LIN {X 0,Y 375.925,Z 316.158,A -85,B 0,C 180,E1 -12375.269,E2 -12375.269} C_VEL
LIN {X 0,Y 375.933,Z 316.15,A -85,B 0,C 180,E1 -12378.4,E2 -12378.4} C_VEL
LIN {X 0,Y 375.971,Z 316.15,A -85,B 0,C 180,E1 -12381.73,E2 -12381.73} C_VEL
LIN {X 0,Y 375.979,Z 316.144,A -85,B 0,C 180,E1 -12385.333,E2 -12385.333} C_VEL
LIN {X 0,Y 375.957,Z 316.149,A -85,B 0,C 180,E1 -12388.438,E2 -12388.438} C_VEL
LIN {X 0,Y 375.983,Z 316.148,A -85,B 0,C 180,E1 -12392.141,E2 -12392.141} C_VEL
LIN {X 0,Y 376.006,Z 316.148,A -85,B 0,C 180,E1 -12394.539,E2 -12394.539} C_VEL
LIN {X 0,Y 375.963,Z 316.147,A -85,B 0,C 180,E1 -12398.046,E2 -12398.046} C_VEL
LIN {X 0,Y 376.024,Z 316.138,A -85,B 0,C 180,E1 -12401.474,E2 -12401.474} C_VEL
LIN {X 0,Y 376.059,Z 316.138,A -85,B 0,C 180,E1 -12404.833,E2 -12404.833} C_VEL
LIN {X 0,Y 376.052,Z 316.142,A -85,B 0,C 180,E1 -12408.137,E2 -12408.137} C_VEL
LIN {X 0,Y 376.259,Z 316.11,A -85,B 0,C 180,E1 -12411.877,E2 -12411.877} C_VEL
LIN {X 0,Y 376.173,Z 316.121,A -85,B 0,C 180,E1 -12414.64,E2 -12414.64} C_VEL
LIN {X 0,Y 376.355,Z 316.102,A -85,B 0,C 180,E1 -12417.86,E2 -12417.86} C_VEL
LIN {X 0,Y 376.491,Z 316.083,A -85,B 0,C 180,E1 -12420,E2 -12420} C_VEL
LIN {X 0,Y 376.19,Z 316.122,A -85,B 0,C 180,E1 -12423.213,E2 -12423.213} C_VEL
LIN {X 0,Y 376.238,Z 316.115,A -85,B 0,C 180,E1 -12426.605,E2 -12426.605} C_VEL
LIN {X 0,Y 376.207,Z 316.119,A -85,B 0,C 180,E1 -12428.595,E2 -12428.595} C_VEL
LIN {X 0,Y 376.052,Z 316.137,A -85,B 0,C 180,E1 -12431.864,E2 -12431.864} C_VEL
LIN {X 0,Y 376.06,Z 316.141,A -85,B 0,C 180,E1 -12435.168,E2 -12435.168} C_VEL
LIN {X 0,Y 376.01,Z 316.143,A -85,B 0,C 180,E1 -12438.527,E2 -12438.527} C_VEL
LIN {X 0,Y 375.958,Z 316.153,A -85,B 0,C 180,E1 -12441.955,E2 -12441.955} C_VEL
LIN {X 0,Y 375.978,Z 316.15,A -85,B 0,C 180,E1 -12445.463,E2 -12445.463} C_VEL
LIN {X 0,Y 375.958,Z 316.156,A -85,B 0,C 180,E1 -12449.08,E2 -12449.08} C_VEL
LIN {X 0,Y 375.95,Z 316.158,A -85,B 0,C 180,E1 -12452.829,E2 -12452.829} C_VEL
LIN {X 0,Y 375.958,Z 316.155,A -85,B 0,C 180,E1 -12455.416,E2 -12455.416} C_VEL
LIN {X 0,Y 375.975,Z 316.15,A -85,B 0,C 180,E1 -12458.271,E2 -12458.271} C_VEL
LIN {X 0,Y 376.009,Z 316.268,A -85,B 0,C 180,E1 -12459.974,E2 -12459.974} C_VEL
LIN {X 0,Y 378.221,Z 326.76,A -85,B 0,C 180,E1 -12462.706,E2 -12462.706} C_VEL
LIN {X 0,Y 378.98,Z 330.682,A -85,B 0,C 180,E1 -12463.678,E2 -12463.678} C_VEL
LIN {X 0,Y 378.967,Z 334.995,A -85,B 0,C 180,E1 -12464.597,E2 -12464.597} C_VEL
LIN {X 0,Y 383.33,Z 356.245,A -85,B 0,C 180,E1 -12465.33,E2 -12465.33} C_VEL
LIN {X 0,Y 384.181,Z 362.884,A -85,B 0,C 180,E1 -12465.516,E2 -12465.516} C_VEL
LIN {X 0,Y 382.729,Z 441.201,A -85,B 0,C 180,E1 -12467.044,E2 -12467.044} C_VEL
LIN {X 0,Y 382.323,Z 451.45,A -85,B 0,C 180,E1 -12467.361,E2 -12467.361} C_VEL
LIN {X 0,Y 381.894,Z 461.344,A -85,B 0,C 180,E1 -12467.801,E2 -12467.801} C_VEL
LIN {X 0,Y 381.198,Z 471.819,A -85,B 0,C 180,E1 -12468.416,E2 -12468.416} C_VEL
LIN {X 0,Y 380.503,Z 481.268,A -85,B 0,C 180,E1 -12469.119,E2 -12469.119} C_VEL
LIN {X 0,Y 379.709,Z 490.561,A -85,B 0,C 180,E1 -12469.97,E2 -12469.97} C_VEL
LIN {X 0,Y 378.669,Z 500.677,A -85,B 0,C 180,E1 -12471.115,E2 -12471.115} C_VEL
LIN {X 0,Y 377.901,Z 508.256,A -85,B 0,C 180,E1 -12472.141,E2 -12472.141} C_VEL
LIN {X 0,Y 377.111,Z 515.955,A -85,B 0,C 180,E1 -12473.39,E2 -12473.39} C_VEL
LIN {X 0,Y 376.23,Z 524.101,A -85,B 0,C 180,E1 -12475.019,E2 -12475.019} C_VEL
LIN {X 0,Y 375.749,Z 529.029,A -85,B 0,C 180,E1 -12476.19,E2 -12476.19} C_VEL
LIN {X 0,Y 375.202,Z 534.748,A -85,B 0,C 180,E1 -12477.882,E2 -12477.882} C_VEL
LIN {X 0,Y 374.831,Z 539.238,A -85,B 0,C 180,E1 -12479.598,E2 -12479.598} C_VEL
LIN {X 0,Y 374.655,Z 541.781,A -85,B 0,C 180,E1 -12480.809,E2 -12480.809} C_VEL
LIN {X 0,Y 374.469,Z 543.607,A -85,B 0,C 180,E1 -12482.018,E2 -12482.018} C_VEL
LIN {X 0,Y 374.226,Z 545.847,A -85,B 0,C 180,E1 -12484.349,E2 -12484.349} C_VEL
LIN {X 0,Y 374.166,Z 546.21,A -85,B 0,C 180,E1 -12485.592,E2 -12485.592} C_VEL
LIN {X 0,Y 374.215,Z 545.984,A -85,B 0,C 180,E1 -12486.963,E2 -12486.963} C_VEL
LIN {X 0,Y 374.245,Z 545.511,A -85,B 0,C 180,E1 -12487.94,E2 -12487.94} C_VEL
LIN {X 0,Y 374.428,Z 543.566,A -85,B 0,C 180,E1 -12489.801,E2 -12489.801} C_VEL
LIN {X 0,Y 374.643,Z 540.922,A -85,B 0,C 180,E1 -12491.403,E2 -12491.403} C_VEL
LIN {X 0,Y 374.892,Z 537.413,A -85,B 0,C 180,E1 -12492.957,E2 -12492.957} C_VEL
LIN {X 0,Y 375.172,Z 533.777,A -85,B 0,C 180,E1 -12494.239,E2 -12494.239} C_VEL
LIN {X 0,Y 375.665,Z 527.744,A -85,B 0,C 180,E1 -12495.924,E2 -12495.924} C_VEL
LIN {X 0,Y 376.402,Z 520.097,A -85,B 0,C 180,E1 -12497.601,E2 -12497.601} C_VEL
LIN {X 0,Y 377.122,Z 512.342,A -85,B 0,C 180,E1 -12498.988,E2 -12498.988} C_VEL
LIN {X 0,Y 377.905,Z 504.742,A -85,B 0,C 180,E1 -12500.122,E2 -12500.122} C_VEL
LIN {X 0,Y 378.638,Z 496.199,A -85,B 0,C 180,E1 -12501.192,E2 -12501.192} C_VEL
LIN {X 0,Y 379.538,Z 486.88,A -85,B 0,C 180,E1 -12502.151,E2 -12502.151} C_VEL
LIN {X 0,Y 380.257,Z 477.25,A -85,B 0,C 180,E1 -12502.967,E2 -12502.967} C_VEL
LIN {X 0,Y 380.884,Z 467.314,A -85,B 0,C 180,E1 -12503.644,E2 -12503.644} C_VEL
LIN {X 0,Y 381.489,Z 455.363,A -85,B 0,C 180,E1 -12504.254,E2 -12504.254} C_VEL
LIN {X 0,Y 381.984,Z 444.529,A -85,B 0,C 180,E1 -12504.64,E2 -12504.64} C_VEL
LIN {X 0,Y 382.331,Z 427.037,A -85,B 0,C 180,E1 -12505.025,E2 -12505.025} C_VEL
LIN {X 0,Y 383.365,Z 360.957,A -85,B 0,C 180,E1 -12506.285,E2 -12506.285} C_VEL
LIN {X 0,Y 379.739,Z 341.554,A -85,B 0,C 180,E1 -12506.864,E2 -12506.864} C_VEL
LIN {X 0,Y 378.777,Z 338.239,A -85,B 0,C 180,E1 -12507.067,E2 -12507.067} C_VEL
LIN {X 0,Y 377.196,Z 334.864,A -85,B 0,C 180,E1 -12507.503,E2 -12507.503} C_VEL
LIN {X 0,Y 374.754,Z 331.16,A -85,B 0,C 180,E1 -12508.331,E2 -12508.331} C_VEL
LIN {X 0,Y 371.314,Z 325.692,A -85,B 0,C 180,E1 -12509.995,E2 -12509.995} C_VEL
LIN {X 0,Y 370.628,Z 323.671,A -85,B 0,C 180,E1 -12510.575,E2 -12510.575} C_VEL
LIN {X 0,Y 369.258,Z 317.027,A -85,B 0,C 180,E1 -12512.523,E2 -12512.523} C_VEL
LIN {X 0,Y 369.189,Z 316.994,A -85,B 0,C 180,E1 -12516.559,E2 -12516.559} C_VEL
LIN {X 0,Y 369.065,Z 317.013,A -85,B 0,C 180,E1 -12519.868,E2 -12519.868} C_VEL
LIN {X 0,Y 369.039,Z 317.019,A -85,B 0,C 180,E1 -12523.772,E2 -12523.772} C_VEL
LIN {X 0,Y 369.003,Z 317.022,A -85,B 0,C 180,E1 -12527.768,E2 -12527.768} C_VEL
LIN {X 0,Y 368.912,Z 317.029,A -85,B 0,C 180,E1 -12531.221,E2 -12531.221} C_VEL
LIN {X 0,Y 368.957,Z 317.026,A -85,B 0,C 180,E1 -12534.776,E2 -12534.776} C_VEL
LIN {X 0,Y 368.965,Z 317.018,A -85,B 0,C 180,E1 -12537.203,E2 -12537.203} C_VEL
LIN {X 0,Y 368.931,Z 317.029,A -85,B 0,C 180,E1 -12540.954,E2 -12540.954} C_VEL
LIN {X 0,Y 368.93,Z 317.014,A -85,B 0,C 180,E1 -12545.001,E2 -12545.001} C_VEL
LIN {X 0,Y 368.91,Z 317.028,A -85,B 0,C 180,E1 -12548.64,E2 -12548.64} C_VEL
LIN {X 0,Y 368.883,Z 317.019,A -85,B 0,C 180,E1 -12552.009,E2 -12552.009} C_VEL
LIN {X 0,Y 368.885,Z 317.032,A -85,B 0,C 180,E1 -12555.176,E2 -12555.176} C_VEL
LIN {X 0,Y 368.875,Z 317.03,A -85,B 0,C 180,E1 -12558.176,E2 -12558.176} C_VEL
LIN {X 0,Y 368.883,Z 317.019,A -85,B 0,C 180,E1 -12561.365,E2 -12561.365} C_VEL
LIN {X 0,Y 368.938,Z 317.028,A -85,B 0,C 180,E1 -12565.146,E2 -12565.146} C_VEL
LIN {X 0,Y 368.931,Z 317.015,A -85,B 0,C 180,E1 -12569.046,E2 -12569.046} C_VEL
LIN {X 0,Y 368.879,Z 317.023,A -85,B 0,C 180,E1 -12572.79,E2 -12572.79} C_VEL
LIN {X 0,Y 368.935,Z 317.029,A -85,B 0,C 180,E1 -12576.117,E2 -12576.117} C_VEL
LIN {X 0,Y 368.939,Z 317.013,A -85,B 0,C 180,E1 -12579.947,E2 -12579.947} C_VEL
LIN {X 0,Y 368.971,Z 317.006,A -85,B 0,C 180,E1 -12583.398,E2 -12583.398} C_VEL
LIN {X 0,Y 369.06,Z 317.009,A -85,B 0,C 180,E1 -12586.79,E2 -12586.79} C_VEL
LIN {X 0,Y 369.064,Z 317.002,A -85,B 0,C 180,E1 -12590.131,E2 -12590.131} C_VEL
LIN {X 0,Y 369.161,Z 316.972,A -85,B 0,C 180,E1 -12593.441,E2 -12593.441} C_VEL
LIN {X 0,Y 369.304,Z 316.976,A -85,B 0,C 180,E1 -12597.818,E2 -12597.818} C_VEL
LIN {X 0,Y 369.237,Z 316.983,A -85,B 0,C 180,E1 -12601.09,E2 -12601.09} C_VEL
LIN {X 0,Y 369.303,Z 316.976,A -85,B 0,C 180,E1 -12602.181,E2 -12602.181} C_VEL
LIN {X 0,Y 369.181,Z 316.979,A -85,B 0,C 180,E1 -12606.558,E2 -12606.558} C_VEL
LIN {X 0,Y 369.064,Z 317.01,A -85,B 0,C 180,E1 -12609.868,E2 -12609.868} C_VEL
LIN {X 0,Y 369.039,Z 316.998,A -85,B 0,C 180,E1 -12613.772,E2 -12613.772} C_VEL
LIN {X 0,Y 368.954,Z 317.019,A -85,B 0,C 180,E1 -12617.744,E2 -12617.744} C_VEL
LIN {X 0,Y 368.91,Z 317.026,A -85,B 0,C 180,E1 -12621.22,E2 -12621.22} C_VEL
LIN {X 0,Y 368.923,Z 317.018,A -85,B 0,C 180,E1 -12624.777,E2 -12624.777} C_VEL
LIN {X 0,Y 368.893,Z 317.035,A -85,B 0,C 180,E1 -12628.792,E2 -12628.792} C_VEL
LIN {X 0,Y 368.897,Z 317.023,A -85,B 0,C 180,E1 -12632.238,E2 -12632.238} C_VEL
LIN {X 0,Y 368.927,Z 317.029,A -85,B 0,C 180,E1 -12635.001,E2 -12635.001} C_VEL
LIN {X 0,Y 368.875,Z 317.031,A -85,B 0,C 180,E1 -12638.633,E2 -12638.633} C_VEL
LIN {X 0,Y 368.856,Z 317.033,A -85,B 0,C 180,E1 -12642.005,E2 -12642.005} C_VEL
LIN {X 0,Y 368.871,Z 317.033,A -85,B 0,C 180,E1 -12645.174,E2 -12645.174} C_VEL
LIN {X 0,Y 368.858,Z 317.038,A -85,B 0,C 180,E1 -12648.174,E2 -12648.174} C_VEL
LIN {X 0,Y 368.875,Z 317.034,A -85,B 0,C 180,E1 -12651.366,E2 -12651.366} C_VEL
LIN {X 0,Y 368.929,Z 317.03,A -85,B 0,C 180,E1 -12655.145,E2 -12655.145} C_VEL
LIN {X 0,Y 368.911,Z 317.028,A -85,B 0,C 180,E1 -12659.045,E2 -12659.045} C_VEL
LIN {X 0,Y 368.922,Z 317.065,A -85,B 0,C 180,E1 -12661.436,E2 -12661.436} C_VEL
LIN {X 0,Y 369.725,Z 320.883,A -85,B 0,C 180,E1 -12662.551,E2 -12662.551} C_VEL
LIN {X 0,Y 372.093,Z 333.056,A -85,B 0,C 180,E1 -12665.744,E2 -12665.744} C_VEL
LIN {X 0,Y 372.19,Z 336.68,A -85,B 0,C 180,E1 -12666.638,E2 -12666.638} C_VEL
LIN {X 0,Y 371.462,Z 345.045,A -85,B 0,C 180,E1 -12668.565,E2 -12668.565} C_VEL
LIN {X 0,Y 376.368,Z 374.14,A -85,B 0,C 180,E1 -12669.45,E2 -12669.45} C_VEL
LIN {X 0,Y 375.41,Z 443.445,A -85,B 0,C 180,E1 -12670.805,E2 -12670.805} C_VEL
LIN {X 0,Y 374.992,Z 459.033,A -85,B 0,C 180,E1 -12671.208,E2 -12671.208} C_VEL
LIN {X 0,Y 374.213,Z 471.284,A -85,B 0,C 180,E1 -12671.735,E2 -12671.735} C_VEL
LIN {X 0,Y 373.661,Z 481.522,A -85,B 0,C 180,E1 -12672.345,E2 -12672.345} C_VEL
LIN {X 0,Y 372.753,Z 492.128,A -85,B 0,C 180,E1 -12673.149,E2 -12673.149} C_VEL
LIN {X 0,Y 371.932,Z 502.076,A -85,B 0,C 180,E1 -12674.098,E2 -12674.098} C_VEL
LIN {X 0,Y 371.073,Z 511.172,A -85,B 0,C 180,E1 -12675.155,E2 -12675.155} C_VEL
LIN {X 0,Y 370.312,Z 519.206,A -85,B 0,C 180,E1 -12676.277,E2 -12676.277} C_VEL
LIN {X 0,Y 369.503,Z 527.325,A -85,B 0,C 180,E1 -12677.644,E2 -12677.644} C_VEL
LIN {X 0,Y 368.779,Z 534.078,A -85,B 0,C 180,E1 -12679.014,E2 -12679.014} C_VEL
LIN {X 0,Y 368.379,Z 538.745,A -85,B 0,C 180,E1 -12680.113,E2 -12680.113} C_VEL
LIN {X 0,Y 367.913,Z 544.422,A -85,B 0,C 180,E1 -12681.763,E2 -12681.763} C_VEL
LIN {X 0,Y 367.624,Z 548.89,A -85,B 0,C 180,E1 -12683.413,E2 -12683.413} C_VEL
LIN {X 0,Y 367.488,Z 551.209,A -85,B 0,C 180,E1 -12684.513,E2 -12684.513} C_VEL
LIN {X 0,Y 367.348,Z 554.67,A -85,B 0,C 180,E1 -12686.71,E2 -12686.71} C_VEL
LIN {X 0,Y 367.345,Z 556.31,A -85,B 0,C 180,E1 -12688.904,E2 -12688.904} C_VEL
LIN {X 0,Y 367.369,Z 556.628,A -85,B 0,C 180,E1 -12690,E2 -12690} C_VEL
LIN {X 0,Y 367.312,Z 555.904,A -85,B 0,C 180,E1 -12692.193,E2 -12692.193} C_VEL
LIN {X 0,Y 367.351,Z 554.929,A -85,B 0,C 180,E1 -12693.29,E2 -12693.29} C_VEL
LIN {X 0,Y 367.514,Z 551.83,A -85,B 0,C 180,E1 -12695.487,E2 -12695.487} C_VEL
LIN {X 0,Y 367.697,Z 548.302,A -85,B 0,C 180,E1 -12697.137,E2 -12697.137} C_VEL
LIN {X 0,Y 368.077,Z 543.676,A -85,B 0,C 180,E1 -12698.786,E2 -12698.786} C_VEL
LIN {X 0,Y 368.652,Z 537.8,A -85,B 0,C 180,E1 -12700.434,E2 -12700.434} C_VEL
LIN {X 0,Y 369.38,Z 530.442,A -85,B 0,C 180,E1 -12702.081,E2 -12702.081} C_VEL
LIN {X 0,Y 370.261,Z 522.998,A -85,B 0,C 180,E1 -12703.445,E2 -12703.445} C_VEL
LIN {X 0,Y 371.091,Z 515.106,A -85,B 0,C 180,E1 -12704.655,E2 -12704.655} C_VEL
LIN {X 0,Y 371.993,Z 506.465,A -85,B 0,C 180,E1 -12705.758,E2 -12705.758} C_VEL
LIN {X 0,Y 372.838,Z 497.564,A -85,B 0,C 180,E1 -12706.706,E2 -12706.706} C_VEL
LIN {X 0,Y 373.878,Z 486.51,A -85,B 0,C 180,E1 -12707.644,E2 -12707.644} C_VEL
LIN {X 0,Y 374.673,Z 476.626,A -85,B 0,C 180,E1 -12708.312,E2 -12708.312} C_VEL
LIN {X 0,Y 375.392,Z 465.654,A -85,B 0,C 180,E1 -12708.877,E2 -12708.877} C_VEL
LIN {X 0,Y 375.96,Z 454.848,A -85,B 0,C 180,E1 -12709.272,E2 -12709.272} C_VEL
LIN {X 0,Y 376.343,Z 437.6,A -85,B 0,C 180,E1 -12709.663,E2 -12709.663} C_VEL
LIN {X 0,Y 377.26,Z 374.153,A -85,B 0,C 180,E1 -12710.916,E2 -12710.916} C_VEL
LIN {X 0,Y 372.87,Z 349.586,A -85,B 0,C 180,E1 -12711.71,E2 -12711.71} C_VEL
LIN {X 0,Y 371.857,Z 344.362,A -85,B 0,C 180,E1 -12711.94,E2 -12711.94} C_VEL
LIN {X 0,Y 372.591,Z 335.605,A -85,B 0,C 180,E1 -12713.925,E2 -12713.925} C_VEL
LIN {X 0,Y 370.858,Z 325.957,A -85,B 0,C 180,E1 -12716.403,E2 -12716.403} C_VEL
LIN {X 0,Y 368.916,Z 317.18,A -85,B 0,C 180,E1 -12718.8,E2 -12718.8} C_VEL
LIN {X 0,Y 368.896,Z 317.032,A -85,B 0,C 180,E1 -12722.238,E2 -12722.238} C_VEL
LIN {X 0,Y 368.927,Z 317.032,A -85,B 0,C 180,E1 -12725.002,E2 -12725.002} C_VEL
LIN {X 0,Y 368.904,Z 317.035,A -85,B 0,C 180,E1 -12728.64,E2 -12728.64} C_VEL
LIN {X 0,Y 368.872,Z 317.035,A -85,B 0,C 180,E1 -12732.008,E2 -12732.008} C_VEL
LIN {X 0,Y 368.878,Z 317.037,A -85,B 0,C 180,E1 -12735.176,E2 -12735.176} C_VEL
LIN {X 0,Y 368.881,Z 317.03,A -85,B 0,C 180,E1 -12738.178,E2 -12738.178} C_VEL
LIN {X 0,Y 368.906,Z 317.03,A -85,B 0,C 180,E1 -12741.36,E2 -12741.36} C_VEL
LIN {X 0,Y 368.936,Z 317.02,A -85,B 0,C 180,E1 -12745.147,E2 -12745.147} C_VEL
LIN {X 0,Y 368.928,Z 317.024,A -85,B 0,C 180,E1 -12749.047,E2 -12749.047} C_VEL
LIN {X 0,Y 368.963,Z 317.02,A -85,B 0,C 180,E1 -12752.797,E2 -12752.797} C_VEL
LIN {X 0,Y 368.945,Z 317.023,A -85,B 0,C 180,E1 -12756.113,E2 -12756.113} C_VEL
LIN {X 0,Y 368.937,Z 317.025,A -85,B 0,C 180,E1 -12759.947,E2 -12759.947} C_VEL
LIN {X 0,Y 368.977,Z 317.024,A -85,B 0,C 180,E1 -12763.399,E2 -12763.399} C_VEL
LIN {X 0,Y 369.058,Z 317.003,A -85,B 0,C 180,E1 -12766.791,E2 -12766.791} C_VEL
LIN {X 0,Y 369.069,Z 317.005,A -85,B 0,C 180,E1 -12770.132,E2 -12770.132} C_VEL
LIN {X 0,Y 369.19,Z 316.997,A -85,B 0,C 180,E1 -12772.343,E2 -12772.343} C_VEL
LIN {X 0,Y 369.146,Z 316.998,A -85,B 0,C 180,E1 -12774.538,E2 -12774.538} C_VEL
LIN {X 0,Y 369.32,Z 316.978,A -85,B 0,C 180,E1 -12777.819,E2 -12777.819} C_VEL
LIN {X 0,Y 369.46,Z 316.958,A -85,B 0,C 180,E1 -12780,E2 -12780} C_VEL
LIN {X 0,Y 369.32,Z 316.978,A -85,B 0,C 180,E1 -12782.181,E2 -12782.181} C_VEL
LIN {X 0,Y 369.208,Z 316.992,A -85,B 0,C 180,E1 -12786.592,E2 -12786.592} C_VEL
LIN {X 0,Y 369.139,Z 316.999,A -85,B 0,C 180,E1 -12788.761,E2 -12788.761} C_VEL
LIN {X 0,Y 369.007,Z 317.013,A -85,B 0,C 180,E1 -12792.093,E2 -12792.093} C_VEL
LIN {X 0,Y 368.999,Z 317.02,A -85,B 0,C 180,E1 -12795.465,E2 -12795.465} C_VEL
LIN {X 0,Y 368.96,Z 317.02,A -85,B 0,C 180,E1 -12798.894,E2 -12798.894} C_VEL
LIN {X 0,Y 368.923,Z 317.03,A -85,B 0,C 180,E1 -12802.396,E2 -12802.396} C_VEL
LIN {X 0,Y 368.962,Z 317.026,A -85,B 0,C 180,E1 -12805.983,E2 -12805.983} C_VEL
LIN {X 0,Y 368.944,Z 317.024,A -85,B 0,C 180,E1 -12808.807,E2 -12808.807} C_VEL
LIN {X 0,Y 368.899,Z 317.031,A -85,B 0,C 180,E1 -12812.238,E2 -12812.238} C_VEL
LIN {X 0,Y 368.93,Z 317.029,A -85,B 0,C 180,E1 -12815.002,E2 -12815.002} C_VEL
LIN {X 0,Y 368.912,Z 317.03,A -85,B 0,C 180,E1 -12818.641,E2 -12818.641} C_VEL
LIN {X 0,Y 368.98,Z 317.254,A -85,B 0,C 180,E1 -12819.649,E2 -12819.649} C_VEL
LIN {X 0,Y 371.215,Z 327.729,A -85,B 0,C 180,E1 -12822.408,E2 -12822.408} C_VEL
LIN {X 0,Y 372.128,Z 333.344,A -85,B 0,C 180,E1 -12823.813,E2 -12823.813} C_VEL
LIN {X 0,Y 372.155,Z 335.145,A -85,B 0,C 180,E1 -12824.158,E2 -12824.158} C_VEL
LIN {X 0,Y 376.778,Z 357.392,A -85,B 0,C 180,E1 -12824.949,E2 -12824.949} C_VEL
LIN {X 0,Y 377.575,Z 364.271,A -85,B 0,C 180,E1 -12825.142,E2 -12825.142} C_VEL
LIN {X 0,Y 376.088,Z 441.078,A -85,B 0,C 180,E1 -12826.667,E2 -12826.667} C_VEL
LIN {X 0,Y 375.682,Z 450.833,A -85,B 0,C 180,E1 -12826.964,E2 -12826.964} C_VEL
LIN {X 0,Y 375.204,Z 461.645,A -85,B 0,C 180,E1 -12827.453,E2 -12827.453} C_VEL
LIN {X 0,Y 374.499,Z 471.624,A -85,B 0,C 180,E1 -12828.045,E2 -12828.045} C_VEL
LIN {X 0,Y 373.69,Z 481.951,A -85,B 0,C 180,E1 -12828.834,E2 -12828.834} C_VEL
LIN {X 0,Y 372.786,Z 491.886,A -85,B 0,C 180,E1 -12829.782,E2 -12829.782} C_VEL
LIN {X 0,Y 371.846,Z 500.671,A -85,B 0,C 180,E1 -12830.797,E2 -12830.797} C_VEL
LIN {X 0,Y 370.924,Z 509.201,A -85,B 0,C 180,E1 -12831.991,E2 -12831.991} C_VEL
LIN {X 0,Y 370.106,Z 516.757,A -85,B 0,C 180,E1 -12833.262,E2 -12833.262} C_VEL
LIN {X 0,Y 369.286,Z 524.062,A -85,B 0,C 180,E1 -12834.753,E2 -12834.753} C_VEL
LIN {X 0,Y 368.707,Z 529.598,A -85,B 0,C 180,E1 -12836.114,E2 -12836.114} C_VEL
LIN {X 0,Y 368.192,Z 534.815,A -85,B 0,C 180,E1 -12837.693,E2 -12837.693} C_VEL
LIN {X 0,Y 367.783,Z 539.033,A -85,B 0,C 180,E1 -12839.307,E2 -12839.307} C_VEL
LIN {X 0,Y 367.566,Z 542.088,A -85,B 0,C 180,E1 -12840.819,E2 -12840.819} C_VEL
LIN {X 0,Y 367.26,Z 544.621,A -85,B 0,C 180,E1 -12842.66,E2 -12842.66} C_VEL
LIN {X 0,Y 367.132,Z 545.87,A -85,B 0,C 180,E1 -12844.122,E2 -12844.122} C_VEL
LIN {X 0,Y 367.101,Z 546.282,A -85,B 0,C 180,E1 -12846.295,E2 -12846.295} C_VEL
LIN {X 0,Y 367.144,Z 545.926,A -85,B 0,C 180,E1 -12847.49,E2 -12847.49} C_VEL
LIN {X 0,Y 367.343,Z 543.661,A -85,B 0,C 180,E1 -12849.856,E2 -12849.856} C_VEL
LIN {X 0,Y 367.586,Z 540.758,A -85,B 0,C 180,E1 -12851.611,E2 -12851.611} C_VEL
LIN {X 0,Y 367.785,Z 538.147,A -85,B 0,C 180,E1 -12852.834,E2 -12852.834} C_VEL
LIN {X 0,Y 368.143,Z 533.493,A -85,B 0,C 180,E1 -12854.498,E2 -12854.498} C_VEL
LIN {X 0,Y 368.773,Z 526.54,A -85,B 0,C 180,E1 -12856.397,E2 -12856.397} C_VEL
LIN {X 0,Y 369.334,Z 521.038,A -85,B 0,C 180,E1 -12857.639,E2 -12857.639} C_VEL
LIN {X 0,Y 370.062,Z 513.447,A -85,B 0,C 180,E1 -12859.052,E2 -12859.052} C_VEL
LIN {X 0,Y 370.962,Z 504.768,A -85,B 0,C 180,E1 -12860.378,E2 -12860.378} C_VEL
LIN {X 0,Y 371.742,Z 496.455,A -85,B 0,C 180,E1 -12861.438,E2 -12861.438} C_VEL
LIN {X 0,Y 372.661,Z 487.172,A -85,B 0,C 180,E1 -12862.414,E2 -12862.414} C_VEL
LIN {X 0,Y 373.416,Z 477.576,A -85,B 0,C 180,E1 -12863.245,E2 -12863.245} C_VEL
LIN {X 0,Y 374.195,Z 466.065,A -85,B 0,C 180,E1 -12864.023,E2 -12864.023} C_VEL
LIN {X 0,Y 374.726,Z 455.366,A -85,B 0,C 180,E1 -12864.573,E2 -12864.573} C_VEL
LIN {X 0,Y 375.214,Z 444.628,A -85,B 0,C 180,E1 -12864.963,E2 -12864.963} C_VEL
LIN {X 0,Y 375.575,Z 427.978,A -85,B 0,C 180,E1 -12865.338,E2 -12865.338} C_VEL
LIN {X 0,Y 376.545,Z 361.075,A -85,B 0,C 180,E1 -12866.641,E2 -12866.641} C_VEL
LIN {X 0,Y 371.717,Z 335.589,A -85,B 0,C 180,E1 -12867.461,E2 -12867.461} C_VEL
LIN {X 0,Y 371.872,Z 332.717,A -85,B 0,C 180,E1 -12868.105,E2 -12868.105} C_VEL
LIN {X 0,Y 371.007,Z 325.74,A -85,B 0,C 180,E1 -12870,E2 -12870} C_VEL
LIN {X 0,Y 370.628,Z 323.671,A -85,B 0,C 180,E1 -12870.575,E2 -12870.575} C_VEL
LIN {X 0,Y 369.5,Z 321.978,A -85,B 0,C 180,E1 -12871.109,E2 -12871.109} C_VEL
LIN {X 0,Y 366.085,Z 319.75,A -85,B 0,C 180,E1 -12871.961,E2 -12871.961} C_VEL
LIN {X 0,Y 362.865,Z 318.218,A -85,B 0,C 180,E1 -12872.869,E2 -12872.869} C_VEL
LIN {X 0,Y 362.047,Z 317.885,A -85,B 0,C 180,E1 -12873.484,E2 -12873.484} C_VEL
LIN {X 0,Y 362.15,Z 317.872,A -85,B 0,C 180,E1 -12876.687,E2 -12876.687} C_VEL
LIN {X 0,Y 362.002,Z 317.892,A -85,B 0,C 180,E1 -12880.063,E2 -12880.063} C_VEL
LIN {X 0,Y 362,Z 317.894,A -85,B 0,C 180,E1 -12883.899,E2 -12883.899} C_VEL
LIN {X 0,Y 361.969,Z 317.896,A -85,B 0,C 180,E1 -12887.939,E2 -12887.939} C_VEL
LIN {X 0,Y 361.883,Z 317.905,A -85,B 0,C 180,E1 -12891.654,E2 -12891.654} C_VEL
LIN {X 0,Y 361.929,Z 317.9,A -85,B 0,C 180,E1 -12895.29,E2 -12895.29} C_VEL
LIN {X 0,Y 361.91,Z 317.892,A -85,B 0,C 180,E1 -12897.779,E2 -12897.779} C_VEL
LIN {X 0,Y 361.839,Z 317.911,A -85,B 0,C 180,E1 -12901.629,E2 -12901.629} C_VEL
LIN {X 0,Y 361.876,Z 317.896,A -85,B 0,C 180,E1 -12905.345,E2 -12905.345} C_VEL
LIN {X 0,Y 361.872,Z 317.904,A -85,B 0,C 180,E1 -12909.027,E2 -12909.027} C_VEL
LIN {X 0,Y 361.837,Z 317.904,A -85,B 0,C 180,E1 -12912.829,E2 -12912.829} C_VEL
LIN {X 0,Y 361.821,Z 317.912,A -85,B 0,C 180,E1 -12915.946,E2 -12915.946} C_VEL
LIN {X 0,Y 361.831,Z 317.895,A -85,B 0,C 180,E1 -12919.246,E2 -12919.246} C_VEL
LIN {X 0,Y 361.867,Z 317.9,A -85,B 0,C 180,E1 -12922.982,E2 -12922.982} C_VEL
LIN {X 0,Y 361.861,Z 317.904,A -85,B 0,C 180,E1 -12926.631,E2 -12926.631} C_VEL
LIN {X 0,Y 361.867,Z 317.885,A -85,B 0,C 180,E1 -12929.671,E2 -12929.671} C_VEL
LIN {X 0,Y 361.881,Z 317.895,A -85,B 0,C 180,E1 -12933.469,E2 -12933.469} C_VEL
LIN {X 0,Y 361.885,Z 317.902,A -85,B 0,C 180,E1 -12937.144,E2 -12937.144} C_VEL
LIN {X 0,Y 361.888,Z 317.88,A -85,B 0,C 180,E1 -12940.722,E2 -12940.722} C_VEL
LIN {X 0,Y 361.945,Z 317.882,A -85,B 0,C 180,E1 -12944.226,E2 -12944.226} C_VEL
LIN {X 0,Y 362.001,Z 317.886,A -85,B 0,C 180,E1 -12946.528,E2 -12946.528} C_VEL
LIN {X 0,Y 362.001,Z 317.883,A -85,B 0,C 180,E1 -12949.937,E2 -12949.937} C_VEL
LIN {X 0,Y 362.124,Z 317.848,A -85,B 0,C 180,E1 -12953.313,E2 -12953.313} C_VEL
LIN {X 0,Y 362.267,Z 317.852,A -85,B 0,C 180,E1 -12957.776,E2 -12957.776} C_VEL
LIN {X 0,Y 362.205,Z 317.859,A -85,B 0,C 180,E1 -12961.112,E2 -12961.112} C_VEL
LIN {X 0,Y 362.266,Z 317.852,A -85,B 0,C 180,E1 -12962.223,E2 -12962.223} C_VEL
LIN {X 0,Y 362.143,Z 317.856,A -85,B 0,C 180,E1 -12966.686,E2 -12966.686} C_VEL
LIN {X 0,Y 362.001,Z 317.889,A -85,B 0,C 180,E1 -12970.063,E2 -12970.063} C_VEL
LIN {X 0,Y 361.981,Z 317.875,A -85,B 0,C 180,E1 -12973.886,E2 -12973.886} C_VEL
LIN {X 0,Y 361.888,Z 317.904,A -85,B 0,C 180,E1 -12978.103,E2 -12978.103} C_VEL
LIN {X 0,Y 361.855,Z 317.906,A -85,B 0,C 180,E1 -12981.655,E2 -12981.655} C_VEL
LIN {X 0,Y 361.88,Z 317.899,A -85,B 0,C 180,E1 -12985.293,E2 -12985.293} C_VEL
LIN {X 0,Y 361.855,Z 317.907,A -85,B 0,C 180,E1 -12989.073,E2 -12989.073} C_VEL
LIN {X 0,Y 361.847,Z 317.905,A -85,B 0,C 180,E1 -12992.944,E2 -12992.944} C_VEL
LIN {X 0,Y 361.866,Z 317.906,A -85,B 0,C 180,E1 -12995.636,E2 -12995.636} C_VEL
LIN {X 0,Y 361.824,Z 317.909,A -85,B 0,C 180,E1 -12999.017,E2 -12999.017} C_VEL
LIN {X 0,Y 361.827,Z 317.908,A -85,B 0,C 180,E1 -13002.83,E2 -13002.83} C_VEL
LIN {X 0,Y 361.811,Z 317.915,A -85,B 0,C 180,E1 -13005.947,E2 -13005.947} C_VEL
LIN {X 0,Y 361.808,Z 317.914,A -85,B 0,C 180,E1 -13009.249,E2 -13009.249} C_VEL
LIN {X 0,Y 361.86,Z 317.913,A -85,B 0,C 180,E1 -13012.981,E2 -13012.981} C_VEL
LIN {X 0,Y 361.856,Z 317.902,A -85,B 0,C 180,E1 -13016.631,E2 -13016.631} C_VEL
LIN {X 0,Y 361.855,Z 317.908,A -85,B 0,C 180,E1 -13019.67,E2 -13019.67} C_VEL
LIN {X 0,Y 361.887,Z 317.99,A -85,B 0,C 180,E1 -13021.154,E2 -13021.154} C_VEL
LIN {X 0,Y 364.186,Z 329.168,A -85,B 0,C 180,E1 -13024.265,E2 -13024.265} C_VEL
LIN {X 0,Y 365.35,Z 336.451,A -85,B 0,C 180,E1 -13026.174,E2 -13026.174} C_VEL
LIN {X 0,Y 364.596,Z 344.812,A -85,B 0,C 180,E1 -13028.151,E2 -13028.151} C_VEL
LIN {X 0,Y 366.874,Z 357.991,A -85,B 0,C 180,E1 -13028.597,E2 -13028.597} C_VEL
LIN {X 0,Y 369.716,Z 375.724,A -85,B 0,C 180,E1 -13029.125,E2 -13029.125} C_VEL
LIN {X 0,Y 368.481,Z 450.989,A -85,B 0,C 180,E1 -13030.647,E2 -13030.647} C_VEL
LIN {X 0,Y 368.152,Z 460.769,A -85,B 0,C 180,E1 -13030.954,E2 -13030.954} C_VEL
LIN {X 0,Y 367.482,Z 470.708,A -85,B 0,C 180,E1 -13031.389,E2 -13031.389} C_VEL
LIN {X 0,Y 366.889,Z 481.052,A -85,B 0,C 180,E1 -13032.008,E2 -13032.008} C_VEL
LIN {X 0,Y 365.947,Z 491.731,A -85,B 0,C 180,E1 -13032.826,E2 -13032.826} C_VEL
LIN {X 0,Y 365.073,Z 501.732,A -85,B 0,C 180,E1 -13033.791,E2 -13033.791} C_VEL
LIN {X 0,Y 364.168,Z 510.869,A -85,B 0,C 180,E1 -13034.867,E2 -13034.867} C_VEL
LIN {X 0,Y 363.367,Z 518.94,A -85,B 0,C 180,E1 -13036.009,E2 -13036.009} C_VEL
LIN {X 0,Y 362.542,Z 527.092,A -85,B 0,C 180,E1 -13037.403,E2 -13037.403} C_VEL
LIN {X 0,Y 361.761,Z 533.87,A -85,B 0,C 180,E1 -13038.798,E2 -13038.798} C_VEL
LIN {X 0,Y 361.346,Z 538.552,A -85,B 0,C 180,E1 -13039.919,E2 -13039.919} C_VEL
LIN {X 0,Y 360.874,Z 544.256,A -85,B 0,C 180,E1 -13041.601,E2 -13041.601} C_VEL
LIN {X 0,Y 360.565,Z 548.743,A -85,B 0,C 180,E1 -13043.284,E2 -13043.284} C_VEL
LIN {X 0,Y 360.406,Z 551.062,A -85,B 0,C 180,E1 -13044.405,E2 -13044.405} C_VEL
LIN {X 0,Y 360.27,Z 554.547,A -85,B 0,C 180,E1 -13046.645,E2 -13046.645} C_VEL
LIN {X 0,Y 360.244,Z 556.204,A -85,B 0,C 180,E1 -13048.882,E2 -13048.882} C_VEL
LIN {X 0,Y 360.27,Z 556.522,A -85,B 0,C 180,E1 -13050,E2 -13050} C_VEL
LIN {X 0,Y 360.219,Z 555.823,A -85,B 0,C 180,E1 -13052.236,E2 -13052.236} C_VEL
LIN {X 0,Y 360.274,Z 554.849,A -85,B 0,C 180,E1 -13053.355,E2 -13053.355} C_VEL
LIN {X 0,Y 360.43,Z 551.773,A -85,B 0,C 180,E1 -13055.595,E2 -13055.595} C_VEL
LIN {X 0,Y 360.629,Z 548.259,A -85,B 0,C 180,E1 -13057.277,E2 -13057.277} C_VEL
LIN {X 0,Y 361.047,Z 543.649,A -85,B 0,C 180,E1 -13058.959,E2 -13058.959} C_VEL
LIN {X 0,Y 361.643,Z 537.796,A -85,B 0,C 180,E1 -13060.639,E2 -13060.639} C_VEL
LIN {X 0,Y 362.426,Z 530.456,A -85,B 0,C 180,E1 -13062.316,E2 -13062.316} C_VEL
LIN {X 0,Y 363.354,Z 523.034,A -85,B 0,C 180,E1 -13063.706,E2 -13063.706} C_VEL
LIN {X 0,Y 364.175,Z 515.525,A -85,B 0,C 180,E1 -13064.89,E2 -13064.89} C_VEL
LIN {X 0,Y 365.162,Z 506.559,A -85,B 0,C 180,E1 -13066.061,E2 -13066.061} C_VEL
LIN {X 0,Y 366.195,Z 496.202,A -85,B 0,C 180,E1 -13067.162,E2 -13067.162} C_VEL
LIN {X 0,Y 367.137,Z 486.704,A -85,B 0,C 180,E1 -13067.979,E2 -13067.979} C_VEL
LIN {X 0,Y 367.961,Z 476.906,A -85,B 0,C 180,E1 -13068.658,E2 -13068.658} C_VEL
LIN {X 0,Y 368.747,Z 465.261,A -85,B 0,C 180,E1 -13069.266,E2 -13069.266} C_VEL
LIN {X 0,Y 369.364,Z 454.315,A -85,B 0,C 180,E1 -13069.666,E2 -13069.666} C_VEL
LIN {X 0,Y 369.776,Z 435.562,A -85,B 0,C 180,E1 -13070.093,E2 -13070.093} C_VEL
LIN {X 0,Y 370.747,Z 375.443,A -85,B 0,C 180,E1 -13071.301,E2 -13071.301} C_VEL
LIN {X 0,Y 366.489,Z 351.417,A -85,B 0,C 180,E1 -13072.099,E2 -13072.099} C_VEL
LIN {X 0,Y 365.087,Z 344.379,A -85,B 0,C 180,E1 -13072.384,E2 -13072.384} C_VEL
LIN {X 0,Y 365.658,Z 338.092,A -85,B 0,C 180,E1 -13073.805,E2 -13073.805} C_VEL
LIN {X 0,Y 365.103,Z 333.178,A -85,B 0,C 180,E1 -13075.055,E2 -13075.055} C_VEL
LIN {X 0,Y 362.783,Z 322.138,A -85,B 0,C 180,E1 -13078.02,E2 -13078.02} C_VEL
LIN {X 0,Y 361.865,Z 318.064,A -85,B 0,C 180,E1 -13079.191,E2 -13079.191} C_VEL
LIN {X 0,Y 361.846,Z 317.913,A -85,B 0,C 180,E1 -13082.945,E2 -13082.945} C_VEL
LIN {X 0,Y 361.866,Z 317.909,A -85,B 0,C 180,E1 -13085.637,E2 -13085.637} C_VEL
LIN {X 0,Y 361.864,Z 317.906,A -85,B 0,C 180,E1 -13089.026,E2 -13089.026} C_VEL
LIN {X 0,Y 361.832,Z 317.915,A -85,B 0,C 180,E1 -13092.829,E2 -13092.829} C_VEL
LIN {X 0,Y 361.816,Z 317.913,A -85,B 0,C 180,E1 -13095.947,E2 -13095.947} C_VEL
LIN {X 0,Y 361.834,Z 317.91,A -85,B 0,C 180,E1 -13099.245,E2 -13099.245} C_VEL
LIN {X 0,Y 361.862,Z 317.908,A -85,B 0,C 180,E1 -13102.777,E2 -13102.777} C_VEL
LIN {X 0,Y 361.853,Z 317.906,A -85,B 0,C 180,E1 -13105.72,E2 -13105.72} C_VEL
LIN {X 0,Y 361.872,Z 317.904,A -85,B 0,C 180,E1 -13109.672,E2 -13109.672} C_VEL
LIN {X 0,Y 361.954,Z 317.894,A -85,B 0,C 180,E1 -13113.475,E2 -13113.475} C_VEL
LIN {X 0,Y 361.89,Z 317.9,A -85,B 0,C 180,E1 -13117.145,E2 -13117.145} C_VEL
LIN {X 0,Y 361.921,Z 317.9,A -85,B 0,C 180,E1 -13120.725,E2 -13120.725} C_VEL
LIN {X 0,Y 361.947,Z 317.896,A -85,B 0,C 180,E1 -13124.226,E2 -13124.226} C_VEL
LIN {X 0,Y 361.999,Z 317.882,A -85,B 0,C 180,E1 -13126.528,E2 -13126.528} C_VEL
LIN {X 0,Y 362.032,Z 317.883,A -85,B 0,C 180,E1 -13129.938,E2 -13129.938} C_VEL
LIN {X 0,Y 362.148,Z 317.871,A -85,B 0,C 180,E1 -13132.193,E2 -13132.193} C_VEL
LIN {X 0,Y 362.12,Z 317.874,A -85,B 0,C 180,E1 -13134.432,E2 -13134.432} C_VEL
LIN {X 0,Y 362.284,Z 317.854,A -85,B 0,C 180,E1 -13137.777,E2 -13137.777} C_VEL
LIN {X 0,Y 362.43,Z 317.834,A -85,B 0,C 180,E1 -13140,E2 -13140} C_VEL
LIN {X 0,Y 362.284,Z 317.855,A -85,B 0,C 180,E1 -13142.224,E2 -13142.224} C_VEL
LIN {X 0,Y 362.174,Z 317.87,A -85,B 0,C 180,E1 -13146.686,E2 -13146.686} C_VEL
LIN {X 0,Y 362.075,Z 317.878,A -85,B 0,C 180,E1 -13148.933,E2 -13148.933} C_VEL
LIN {X 0,Y 361.962,Z 317.89,A -85,B 0,C 180,E1 -13152.333,E2 -13152.333} C_VEL
LIN {X 0,Y 361.963,Z 317.895,A -85,B 0,C 180,E1 -13154.621,E2 -13154.621} C_VEL
LIN {X 0,Y 361.957,Z 317.897,A -85,B 0,C 180,E1 -13158.1,E2 -13158.1} C_VEL
LIN {X 0,Y 361.862,Z 317.909,A -85,B 0,C 180,E1 -13161.655,E2 -13161.655} C_VEL
LIN {X 0,Y 361.904,Z 317.903,A -85,B 0,C 180,E1 -13165.292,E2 -13165.292} C_VEL
LIN {X 0,Y 361.895,Z 317.907,A -85,B 0,C 180,E1 -13169.085,E2 -13169.085} C_VEL
LIN {X 0,Y 361.849,Z 317.913,A -85,B 0,C 180,E1 -13172.945,E2 -13172.945} C_VEL
LIN {X 0,Y 361.869,Z 317.908,A -85,B 0,C 180,E1 -13175.637,E2 -13175.637} C_VEL
LIN {X 0,Y 361.889,Z 317.943,A -85,B 0,C 180,E1 -13179.139,E2 -13179.139} C_VEL
LIN {X 0,Y 362.364,Z 320.035,A -85,B 0,C 180,E1 -13179.794,E2 -13179.794} C_VEL
LIN {X 0,Y 364.468,Z 330.042,A -85,B 0,C 180,E1 -13182.447,E2 -13182.447} C_VEL
LIN {X 0,Y 365.279,Z 334.925,A -85,B 0,C 180,E1 -13183.655,E2 -13183.655} C_VEL
LIN {X 0,Y 366.905,Z 341.949,A -85,B 0,C 180,E1 -13183.968,E2 -13183.968} C_VEL
LIN {X 0,Y 370.882,Z 362.439,A -85,B 0,C 180,E1 -13184.675,E2 -13184.675} C_VEL
LIN {X 0,Y 370.496,Z 392.955,A -85,B 0,C 180,E1 -13185.296,E2 -13185.296} C_VEL
LIN {X 0,Y 369.423,Z 441.846,A -85,B 0,C 180,E1 -13186.297,E2 -13186.297} C_VEL
LIN {X 0,Y 369.008,Z 451.787,A -85,B 0,C 180,E1 -13186.619,E2 -13186.619} C_VEL
LIN {X 0,Y 368.505,Z 462.23,A -85,B 0,C 180,E1 -13187.108,E2 -13187.108} C_VEL
LIN {X 0,Y 367.725,Z 472.504,A -85,B 0,C 180,E1 -13187.739,E2 -13187.739} C_VEL
LIN {X 0,Y 366.921,Z 482.424,A -85,B 0,C 180,E1 -13188.519,E2 -13188.519} C_VEL
LIN {X 0,Y 366.05,Z 491.672,A -85,B 0,C 180,E1 -13189.414,E2 -13189.414} C_VEL
LIN {X 0,Y 364.977,Z 501.246,A -85,B 0,C 180,E1 -13190.547,E2 -13190.547} C_VEL
LIN {X 0,Y 364.177,Z 508.164,A -85,B 0,C 180,E1 -13191.511,E2 -13191.511} C_VEL
LIN {X 0,Y 363.318,Z 515.785,A -85,B 0,C 180,E1 -13192.78,E2 -13192.78} C_VEL
LIN {X 0,Y 362.362,Z 523.786,A -85,B 0,C 180,E1 -13194.419,E2 -13194.419} C_VEL
LIN {X 0,Y 361.756,Z 529.064,A -85,B 0,C 180,E1 -13195.709,E2 -13195.709} C_VEL
LIN {X 0,Y 361.286,Z 533.449,A -85,B 0,C 180,E1 -13196.997,E2 -13196.997} C_VEL
LIN {X 0,Y 360.766,Z 538.822,A -85,B 0,C 180,E1 -13198.999,E2 -13198.999} C_VEL
LIN {X 0,Y 360.476,Z 542.386,A -85,B 0,C 180,E1 -13200.83,E2 -13200.83} C_VEL
LIN {X 0,Y 360.248,Z 544.191,A -85,B 0,C 180,E1 -13202.082,E2 -13202.082} C_VEL
LIN {X 0,Y 360.09,Z 545.832,A -85,B 0,C 180,E1 -13203.87,E2 -13203.87} C_VEL
LIN {X 0,Y 360.004,Z 546.473,A -85,B 0,C 180,E1 -13205.798,E2 -13205.798} C_VEL
LIN {X 0,Y 360.027,Z 546.164,A -85,B 0,C 180,E1 -13207.02,E2 -13207.02} C_VEL
LIN {X 0,Y 360.198,Z 544.413,A -85,B 0,C 180,E1 -13209.439,E2 -13209.439} C_VEL
LIN {X 0,Y 360.423,Z 541.799,A -85,B 0,C 180,E1 -13211.232,E2 -13211.232} C_VEL
LIN {X 0,Y 360.746,Z 538.078,A -85,B 0,C 180,E1 -13213.009,E2 -13213.009} C_VEL
LIN {X 0,Y 361.203,Z 532.159,A -85,B 0,C 180,E1 -13215.06,E2 -13215.06} C_VEL
LIN {X 0,Y 361.751,Z 526.867,A -85,B 0,C 180,E1 -13216.519,E2 -13216.519} C_VEL
LIN {X 0,Y 362.384,Z 520.485,A -85,B 0,C 180,E1 -13217.967,E2 -13217.967} C_VEL
LIN {X 0,Y 363.194,Z 512.752,A -85,B 0,C 180,E1 -13219.407,E2 -13219.407} C_VEL
LIN {X 0,Y 364.059,Z 504.667,A -85,B 0,C 180,E1 -13220.655,E2 -13220.655} C_VEL
LIN {X 0,Y 364.838,Z 496.684,A -85,B 0,C 180,E1 -13221.693,E2 -13221.693} C_VEL
LIN {X 0,Y 365.784,Z 487.43,A -85,B 0,C 180,E1 -13222.687,E2 -13222.687} C_VEL
LIN {X 0,Y 366.568,Z 477.966,A -85,B 0,C 180,E1 -13223.525,E2 -13223.525} C_VEL
LIN {X 0,Y 367.291,Z 467.38,A -85,B 0,C 180,E1 -13224.271,E2 -13224.271} C_VEL
LIN {X 0,Y 367.943,Z 455.49,A -85,B 0,C 180,E1 -13224.898,E2 -13224.898} C_VEL
LIN {X 0,Y 368.455,Z 445.208,A -85,B 0,C 180,E1 -13225.282,E2 -13225.282} C_VEL
LIN {X 0,Y 368.862,Z 427.533,A -85,B 0,C 180,E1 -13225.686,E2 -13225.686} C_VEL
LIN {X 0,Y 369.869,Z 362.085,A -85,B 0,C 180,E1 -13226.985,E2 -13226.985} C_VEL
LIN {X 0,Y 365.075,Z 336.857,A -85,B 0,C 180,E1 -13227.794,E2 -13227.794} C_VEL
LIN {X 0,Y 364.885,Z 335.153,A -85,B 0,C 180,E1 -13227.93,E2 -13227.93} C_VEL
LIN {X 0,Y 364.733,Z 331.454,A -85,B 0,C 180,E1 -13228.896,E2 -13228.896} C_VEL
LIN {X 0,Y 363.305,Z 323.631,A -85,B 0,C 180,E1 -13231.109,E2 -13231.109} C_VEL
LIN {X 0,Y 362.198,Z 317.926,A -85,B 0,C 180,E1 -13232.815,E2 -13232.815} C_VEL
LIN {X 0,Y 362.047,Z 317.885,A -85,B 0,C 180,E1 -13233.484,E2 -13233.484} C_VEL
LIN {X 0,Y 361.312,Z 317.979,A -85,B 0,C 180,E1 -13234.413,E2 -13234.413} C_VEL
LIN {X 0,Y 358.511,Z 318.322,A -85,B 0,C 180,E1 -13235.926,E2 -13235.926} C_VEL
LIN {X 0,Y 356.168,Z 318.622,A -85,B 0,C 180,E1 -13237.15,E2 -13237.15} C_VEL
LIN {X 0,Y 355.134,Z 318.743,A -85,B 0,C 180,E1 -13238.095,E2 -13238.095} C_VEL
LIN {X 0,Y 355.031,Z 318.754,A -85,B 0,C 180,E1 -13238.415,E2 -13238.415} C_VEL
LIN {X 0,Y 354.936,Z 318.766,A -85,B 0,C 180,E1 -13241.421,E2 -13241.421} C_VEL
LIN {X 0,Y 354.921,Z 318.77,A -85,B 0,C 180,E1 -13244.917,E2 -13244.917} C_VEL
LIN {X 0,Y 354.903,Z 318.77,A -85,B 0,C 180,E1 -13248.472,E2 -13248.472} C_VEL
LIN {X 0,Y 354.829,Z 318.786,A -85,B 0,C 180,E1 -13252.107,E2 -13252.107} C_VEL
LIN {X 0,Y 354.9,Z 318.774,A -85,B 0,C 180,E1 -13255.828,E2 -13255.828} C_VEL
LIN {X 0,Y 354.819,Z 318.784,A -85,B 0,C 180,E1 -13259.682,E2 -13259.682} C_VEL
LIN {X 0,Y 354.808,Z 318.775,A -85,B 0,C 180,E1 -13263.702,E2 -13263.702} C_VEL
LIN {X 0,Y 354.8,Z 318.786,A -85,B 0,C 180,E1 -13266.459,E2 -13266.459} C_VEL
LIN {X 0,Y 354.826,Z 318.784,A -85,B 0,C 180,E1 -13269.424,E2 -13269.424} C_VEL
LIN {X 0,Y 354.79,Z 318.781,A -85,B 0,C 180,E1 -13272.867,E2 -13272.867} C_VEL
LIN {X 0,Y 354.77,Z 318.792,A -85,B 0,C 180,E1 -13276.104,E2 -13276.104} C_VEL
LIN {X 0,Y 354.783,Z 318.773,A -85,B 0,C 180,E1 -13279.178,E2 -13279.178} C_VEL
LIN {X 0,Y 354.803,Z 318.774,A -85,B 0,C 180,E1 -13282.404,E2 -13282.404} C_VEL
LIN {X 0,Y 354.814,Z 318.785,A -85,B 0,C 180,E1 -13284.941,E2 -13284.941} C_VEL
LIN {X 0,Y 354.795,Z 318.775,A -85,B 0,C 180,E1 -13288.405,E2 -13288.405} C_VEL
LIN {X 0,Y 354.804,Z 318.762,A -85,B 0,C 180,E1 -13291.615,E2 -13291.615} C_VEL
LIN {X 0,Y 354.854,Z 318.778,A -85,B 0,C 180,E1 -13295.423,E2 -13295.423} C_VEL
LIN {X 0,Y 354.829,Z 318.771,A -85,B 0,C 180,E1 -13299.113,E2 -13299.113} C_VEL
LIN {X 0,Y 354.882,Z 318.748,A -85,B 0,C 180,E1 -13302.719,E2 -13302.719} C_VEL
LIN {X 0,Y 354.954,Z 318.763,A -85,B 0,C 180,E1 -13306.255,E2 -13306.255} C_VEL
LIN {X 0,Y 354.957,Z 318.762,A -85,B 0,C 180,E1 -13309.735,E2 -13309.735} C_VEL
LIN {X 0,Y 355.09,Z 318.724,A -85,B 0,C 180,E1 -13313.18,E2 -13313.18} C_VEL
LIN {X 0,Y 355.23,Z 318.728,A -85,B 0,C 180,E1 -13317.732,E2 -13317.732} C_VEL
LIN {X 0,Y 355.174,Z 318.734,A -85,B 0,C 180,E1 -13321.134,E2 -13321.134} C_VEL
LIN {X 0,Y 355.228,Z 318.727,A -85,B 0,C 180,E1 -13322.267,E2 -13322.267} C_VEL
LIN {X 0,Y 355.107,Z 318.734,A -85,B 0,C 180,E1 -13326.819,E2 -13326.819} C_VEL
LIN {X 0,Y 354.957,Z 318.766,A -85,B 0,C 180,E1 -13330.264,E2 -13330.264} C_VEL
LIN {X 0,Y 354.924,Z 318.753,A -85,B 0,C 180,E1 -13334.005,E2 -13334.005} C_VEL
LIN {X 0,Y 354.845,Z 318.781,A -85,B 0,C 180,E1 -13338.069,E2 -13338.069} C_VEL
LIN {X 0,Y 354.808,Z 318.782,A -85,B 0,C 180,E1 -13342.107,E2 -13342.107} C_VEL
LIN {X 0,Y 354.848,Z 318.768,A -85,B 0,C 180,E1 -13344.577,E2 -13344.577} C_VEL
LIN {X 0,Y 354.797,Z 318.788,A -85,B 0,C 180,E1 -13348.385,E2 -13348.385} C_VEL
LIN {X 0,Y 354.786,Z 318.781,A -85,B 0,C 180,E1 -13352.333,E2 -13352.333} C_VEL
LIN {X 0,Y 354.82,Z 318.783,A -85,B 0,C 180,E1 -13355.699,E2 -13355.699} C_VEL
LIN {X 0,Y 354.767,Z 318.791,A -85,B 0,C 180,E1 -13359.412,E2 -13359.412} C_VEL
LIN {X 0,Y 354.779,Z 318.786,A -85,B 0,C 180,E1 -13362.865,E2 -13362.865} C_VEL
LIN {X 0,Y 354.76,Z 318.792,A -85,B 0,C 180,E1 -13366.102,E2 -13366.102} C_VEL
LIN {X 0,Y 354.761,Z 318.792,A -85,B 0,C 180,E1 -13369.175,E2 -13369.175} C_VEL
LIN {X 0,Y 354.798,Z 318.788,A -85,B 0,C 180,E1 -13372.404,E2 -13372.404} C_VEL
LIN {X 0,Y 354.807,Z 318.791,A -85,B 0,C 180,E1 -13374.94,E2 -13374.94} C_VEL
LIN {X 0,Y 354.791,Z 318.791,A -85,B 0,C 180,E1 -13378.405,E2 -13378.405} C_VEL
LIN {X 0,Y 354.839,Z 318.959,A -85,B 0,C 180,E1 -13380.882,E2 -13380.882} C_VEL
LIN {X 0,Y 357.393,Z 331.353,A -85,B 0,C 180,E1 -13384.366,E2 -13384.366} C_VEL
LIN {X 0,Y 358.391,Z 337.423,A -85,B 0,C 180,E1 -13385.989,E2 -13385.989} C_VEL
LIN {X 0,Y 357.745,Z 344.607,A -85,B 0,C 180,E1 -13387.722,E2 -13387.722} C_VEL
LIN {X 0,Y 358.475,Z 349.078,A -85,B 0,C 180,E1 -13387.923,E2 -13387.923} C_VEL
LIN {X 0,Y 363.033,Z 376.629,A -85,B 0,C 180,E1 -13388.772,E2 -13388.772} C_VEL
LIN {X 0,Y 361.725,Z 451.16,A -85,B 0,C 180,E1 -13390.307,E2 -13390.307} C_VEL
LIN {X 0,Y 361.396,Z 460.845,A -85,B 0,C 180,E1 -13390.621,E2 -13390.621} C_VEL
LIN {X 0,Y 360.66,Z 471.339,A -85,B 0,C 180,E1 -13391.097,E2 -13391.097} C_VEL
LIN {X 0,Y 360.133,Z 480.582,A -85,B 0,C 180,E1 -13391.658,E2 -13391.658} C_VEL
LIN {X 0,Y 359.139,Z 491.333,A -85,B 0,C 180,E1 -13392.49,E2 -13392.49} C_VEL
LIN {X 0,Y 358.205,Z 501.386,A -85,B 0,C 180,E1 -13393.471,E2 -13393.471} C_VEL
LIN {X 0,Y 357.318,Z 510.273,A -85,B 0,C 180,E1 -13394.528,E2 -13394.528} C_VEL
LIN {X 0,Y 356.431,Z 518.672,A -85,B 0,C 180,E1 -13395.731,E2 -13395.731} C_VEL
LIN {X 0,Y 355.572,Z 526.853,A -85,B 0,C 180,E1 -13397.152,E2 -13397.152} C_VEL
LIN {X 0,Y 354.757,Z 533.656,A -85,B 0,C 180,E1 -13398.574,E2 -13398.574} C_VEL
LIN {X 0,Y 354.325,Z 538.351,A -85,B 0,C 180,E1 -13399.717,E2 -13399.717} C_VEL
LIN {X 0,Y 353.826,Z 544.082,A -85,B 0,C 180,E1 -13401.433,E2 -13401.433} C_VEL
LIN {X 0,Y 353.501,Z 548.587,A -85,B 0,C 180,E1 -13403.149,E2 -13403.149} C_VEL
LIN {X 0,Y 353.264,Z 552.825,A -85,B 0,C 180,E1 -13405.436,E2 -13405.436} C_VEL
LIN {X 0,Y 353.194,Z 554.419,A -85,B 0,C 180,E1 -13406.578,E2 -13406.578} C_VEL
LIN {X 0,Y 353.143,Z 556.098,A -85,B 0,C 180,E1 -13408.86,E2 -13408.86} C_VEL
LIN {X 0,Y 353.171,Z 556.415,A -85,B 0,C 180,E1 -13410,E2 -13410} C_VEL
LIN {X 0,Y 353.13,Z 555.745,A -85,B 0,C 180,E1 -13412.281,E2 -13412.281} C_VEL
LIN {X 0,Y 353.199,Z 554.77,A -85,B 0,C 180,E1 -13413.422,E2 -13413.422} C_VEL
LIN {X 0,Y 353.336,Z 551.717,A -85,B 0,C 180,E1 -13415.708,E2 -13415.708} C_VEL
LIN {X 0,Y 353.586,Z 548.215,A -85,B 0,C 180,E1 -13417.423,E2 -13417.423} C_VEL
LIN {X 0,Y 354.002,Z 543.621,A -85,B 0,C 180,E1 -13419.139,E2 -13419.139} C_VEL
LIN {X 0,Y 354.793,Z 536.614,A -85,B 0,C 180,E1 -13421.136,E2 -13421.136} C_VEL
LIN {X 0,Y 355.488,Z 530.471,A -85,B 0,C 180,E1 -13422.56,E2 -13422.56} C_VEL
LIN {X 0,Y 356.457,Z 523.07,A -85,B 0,C 180,E1 -13423.976,E2 -13423.976} C_VEL
LIN {X 0,Y 357.395,Z 514.438,A -85,B 0,C 180,E1 -13425.345,E2 -13425.345} C_VEL
LIN {X 0,Y 358.434,Z 505.449,A -85,B 0,C 180,E1 -13426.517,E2 -13426.517} C_VEL
LIN {X 0,Y 359.41,Z 496.381,A -85,B 0,C 180,E1 -13427.496,E2 -13427.496} C_VEL
LIN {X 0,Y 360.403,Z 486.964,A -85,B 0,C 180,E1 -13428.327,E2 -13428.327} C_VEL
LIN {X 0,Y 361.314,Z 476.085,A -85,B 0,C 180,E1 -13429.088,E2 -13429.088} C_VEL
LIN {X 0,Y 362.141,Z 465.006,A -85,B 0,C 180,E1 -13429.669,E2 -13429.669} C_VEL
LIN {X 0,Y 362.769,Z 453.983,A -85,B 0,C 180,E1 -13430.076,E2 -13430.076} C_VEL
LIN {X 0,Y 363.189,Z 435.845,A -85,B 0,C 180,E1 -13430.496,E2 -13430.496} C_VEL
LIN {X 0,Y 364.181,Z 376.176,A -85,B 0,C 180,E1 -13431.719,E2 -13431.719} C_VEL
LIN {X 0,Y 360.094,Z 353.074,A -85,B 0,C 180,E1 -13432.51,E2 -13432.51} C_VEL
LIN {X 0,Y 358.331,Z 344.232,A -85,B 0,C 180,E1 -13432.866,E2 -13432.866} C_VEL
LIN {X 0,Y 358.77,Z 338.161,A -85,B 0,C 180,E1 -13434.291,E2 -13434.291} C_VEL
LIN {X 0,Y 356.932,Z 328.342,A -85,B 0,C 180,E1 -13436.928,E2 -13436.928} C_VEL
LIN {X 0,Y 354.847,Z 319.038,A -85,B 0,C 180,E1 -13439.572,E2 -13439.572} C_VEL
LIN {X 0,Y 354.83,Z 318.786,A -85,B 0,C 180,E1 -13440.336,E2 -13440.336} C_VEL
LIN {X 0,Y 354.804,Z 318.785,A -85,B 0,C 180,E1 -13443.702,E2 -13443.702} C_VEL
LIN {X 0,Y 354.795,Z 318.785,A -85,B 0,C 180,E1 -13446.46,E2 -13446.46} C_VEL
LIN {X 0,Y 354.822,Z 318.78,A -85,B 0,C 180,E1 -13449.424,E2 -13449.424} C_VEL
LIN {X 0,Y 354.784,Z 318.792,A -85,B 0,C 180,E1 -13452.867,E2 -13452.867} C_VEL
LIN {X 0,Y 354.765,Z 318.791,A -85,B 0,C 180,E1 -13456.104,E2 -13456.104} C_VEL
LIN {X 0,Y 354.786,Z 318.787,A -85,B 0,C 180,E1 -13459.179,E2 -13459.179} C_VEL
LIN {X 0,Y 354.805,Z 318.788,A -85,B 0,C 180,E1 -13462.403,E2 -13462.403} C_VEL
LIN {X 0,Y 354.811,Z 318.78,A -85,B 0,C 180,E1 -13464.941,E2 -13464.941} C_VEL
LIN {X 0,Y 354.792,Z 318.785,A -85,B 0,C 180,E1 -13468.405,E2 -13468.405} C_VEL
LIN {X 0,Y 354.846,Z 318.78,A -85,B 0,C 180,E1 -13471.619,E2 -13471.619} C_VEL
LIN {X 0,Y 354.899,Z 318.774,A -85,B 0,C 180,E1 -13474.173,E2 -13474.173} C_VEL
LIN {X 0,Y 354.835,Z 318.78,A -85,B 0,C 180,E1 -13477.894,E2 -13477.894} C_VEL
LIN {X 0,Y 354.923,Z 318.766,A -85,B 0,C 180,E1 -13481.892,E2 -13481.892} C_VEL
LIN {X 0,Y 354.943,Z 318.761,A -85,B 0,C 180,E1 -13485.981,E2 -13485.981} C_VEL
LIN {X 0,Y 354.979,Z 318.765,A -85,B 0,C 180,E1 -13489.736,E2 -13489.736} C_VEL
LIN {X 0,Y 355.129,Z 318.743,A -85,B 0,C 180,E1 -13492.038,E2 -13492.038} C_VEL
LIN {X 0,Y 355.094,Z 318.75,A -85,B 0,C 180,E1 -13494.321,E2 -13494.321} C_VEL
LIN {X 0,Y 355.247,Z 318.73,A -85,B 0,C 180,E1 -13497.733,E2 -13497.733} C_VEL
LIN {X 0,Y 355.399,Z 318.709,A -85,B 0,C 180,E1 -13500,E2 -13500} C_VEL
LIN {X 0,Y 355.247,Z 318.731,A -85,B 0,C 180,E1 -13502.268,E2 -13502.268} C_VEL
LIN {X 0,Y 355.14,Z 318.747,A -85,B 0,C 180,E1 -13506.819,E2 -13506.819} C_VEL
LIN {X 0,Y 355.017,Z 318.757,A -85,B 0,C 180,E1 -13509.113,E2 -13509.113} C_VEL
LIN {X 0,Y 354.923,Z 318.766,A -85,B 0,C 180,E1 -13512.581,E2 -13512.581} C_VEL
LIN {X 0,Y 354.891,Z 318.774,A -85,B 0,C 180,E1 -13516.096,E2 -13516.096} C_VEL
LIN {X 0,Y 354.903,Z 318.773,A -85,B 0,C 180,E1 -13518.472,E2 -13518.472} C_VEL
LIN {X 0,Y 354.816,Z 318.786,A -85,B 0,C 180,E1 -13522.107,E2 -13522.107} C_VEL
LIN {X 0,Y 354.869,Z 318.781,A -85,B 0,C 180,E1 -13525.83,E2 -13525.83} C_VEL
LIN {X 0,Y 354.818,Z 318.787,A -85,B 0,C 180,E1 -13529.682,E2 -13529.682} C_VEL
LIN {X 0,Y 354.807,Z 318.783,A -85,B 0,C 180,E1 -13533.702,E2 -13533.702} C_VEL
LIN {X 0,Y 354.801,Z 318.786,A -85,B 0,C 180,E1 -13536.459,E2 -13536.459} C_VEL
LIN {X 0,Y 354.859,Z 318.924,A -85,B 0,C 180,E1 -13538.78,E2 -13538.78} C_VEL
LIN {X 0,Y 357.075,Z 328.974,A -85,B 0,C 180,E1 -13541.589,E2 -13541.589} C_VEL
LIN {X 0,Y 358.288,Z 335.094,A -85,B 0,C 180,E1 -13543.164,E2 -13543.164} C_VEL
LIN {X 0,Y 359.906,Z 340.936,A -85,B 0,C 180,E1 -13543.451,E2 -13543.451} C_VEL
LIN {X 0,Y 364.176,Z 362.323,A -85,B 0,C 180,E1 -13544.223,E2 -13544.223} C_VEL
LIN {X 0,Y 364.516,Z 364.475,A -85,B 0,C 180,E1 -13544.293,E2 -13544.293} C_VEL
LIN {X 0,Y 362.836,Z 441.591,A -85,B 0,C 180,E1 -13545.882,E2 -13545.882} C_VEL
LIN {X 0,Y 362.393,Z 451.541,A -85,B 0,C 180,E1 -13546.204,E2 -13546.204} C_VEL
LIN {X 0,Y 361.88,Z 462.07,A -85,B 0,C 180,E1 -13546.702,E2 -13546.702} C_VEL
LIN {X 0,Y 361.138,Z 471.801,A -85,B 0,C 180,E1 -13547.3,E2 -13547.3} C_VEL
LIN {X 0,Y 360.314,Z 481.683,A -85,B 0,C 180,E1 -13548.075,E2 -13548.075} C_VEL
LIN {X 0,Y 359.308,Z 491.743,A -85,B 0,C 180,E1 -13549.061,E2 -13549.061} C_VEL
LIN {X 0,Y 358.27,Z 500.576,A -85,B 0,C 180,E1 -13550.112,E2 -13550.112} C_VEL
LIN {X 0,Y 357.271,Z 508.792,A -85,B 0,C 180,E1 -13551.288,E2 -13551.288} C_VEL
LIN {X 0,Y 356.305,Z 516.721,A -85,B 0,C 180,E1 -13552.661,E2 -13552.661} C_VEL
LIN {X 0,Y 355.42,Z 523.894,A -85,B 0,C 180,E1 -13554.167,E2 -13554.167} C_VEL
LIN {X 0,Y 354.712,Z 529.635,A -85,B 0,C 180,E1 -13555.62,E2 -13555.62} C_VEL
LIN {X 0,Y 354.215,Z 534.141,A -85,B 0,C 180,E1 -13556.984,E2 -13556.984} C_VEL
LIN {X 0,Y 353.692,Z 539.045,A -85,B 0,C 180,E1 -13558.894,E2 -13558.894} C_VEL
LIN {X 0,Y 353.469,Z 541.659,A -85,B 0,C 180,E1 -13560.193,E2 -13560.193} C_VEL
LIN {X 0,Y 353.267,Z 543.588,A -85,B 0,C 180,E1 -13561.48,E2 -13561.48} C_VEL
LIN {X 0,Y 353.003,Z 545.786,A -85,B 0,C 180,E1 -13563.626,E2 -13563.626} C_VEL
LIN {X 0,Y 352.892,Z 546.449,A -85,B 0,C 180,E1 -13565.278,E2 -13565.278} C_VEL
LIN {X 0,Y 352.917,Z 546.403,A -85,B 0,C 180,E1 -13566.529,E2 -13566.529} C_VEL
LIN {X 0,Y 352.932,Z 545.987,A -85,B 0,C 180,E1 -13567.769,E2 -13567.769} C_VEL
LIN {X 0,Y 353.076,Z 544.676,A -85,B 0,C 180,E1 -13569.316,E2 -13569.316} C_VEL
LIN {X 0,Y 353.365,Z 541.642,A -85,B 0,C 180,E1 -13571.445,E2 -13571.445} C_VEL
LIN {X 0,Y 353.69,Z 537.828,A -85,B 0,C 180,E1 -13573.255,E2 -13573.255} C_VEL
LIN {X 0,Y 354.131,Z 532.808,A -85,B 0,C 180,E1 -13575.049,E2 -13575.049} C_VEL
LIN {X 0,Y 354.674,Z 527.606,A -85,B 0,C 180,E1 -13576.545,E2 -13576.545} C_VEL
LIN {X 0,Y 355.333,Z 521.393,A -85,B 0,C 180,E1 -13578.014,E2 -13578.014} C_VEL
LIN {X 0,Y 356.152,Z 513.82,A -85,B 0,C 180,E1 -13579.483,E2 -13579.483} C_VEL
LIN {X 0,Y 357.027,Z 506.002,A -85,B 0,C 180,E1 -13580.745,E2 -13580.745} C_VEL
LIN {X 0,Y 357.953,Z 496.905,A -85,B 0,C 180,E1 -13581.959,E2 -13581.959} C_VEL
LIN {X 0,Y 358.93,Z 487.677,A -85,B 0,C 180,E1 -13582.971,E2 -13582.971} C_VEL
LIN {X 0,Y 359.798,Z 477.387,A -85,B 0,C 180,E1 -13583.889,E2 -13583.889} C_VEL
LIN {X 0,Y 360.509,Z 467.601,A -85,B 0,C 180,E1 -13584.59,E2 -13584.59} C_VEL
LIN {X 0,Y 361.185,Z 455.889,A -85,B 0,C 180,E1 -13585.222,E2 -13585.222} C_VEL
LIN {X 0,Y 361.732,Z 444.51,A -85,B 0,C 180,E1 -13585.648,E2 -13585.648} C_VEL
LIN {X 0,Y 362.125,Z 427.755,A -85,B 0,C 180,E1 -13586.036,E2 -13586.036} C_VEL
LIN {X 0,Y 363.224,Z 363.221,A -85,B 0,C 180,E1 -13587.338,E2 -13587.338} C_VEL
LIN {X 0,Y 358.063,Z 335.908,A -85,B 0,C 180,E1 -13588.25,E2 -13588.25} C_VEL
LIN {X 0,Y 357.92,Z 334.235,A -85,B 0,C 180,E1 -13588.594,E2 -13588.594} C_VEL
LIN {X 0,Y 356.925,Z 327.3,A -85,B 0,C 180,E1 -13590.564,E2 -13590.564} C_VEL
LIN {X 0,Y 355.093,Z 318.834,A -85,B 0,C 180,E1 -13593.12,E2 -13593.12} C_VEL
LIN {X 0,Y 355.113,Z 318.75,A -85,B 0,C 180,E1 -13596.82,E2 -13596.82} C_VEL
LIN {X 0,Y 355.031,Z 318.754,A -85,B 0,C 180,E1 -13598.415,E2 -13598.415} C_VEL
LIN {X 0,Y 354.304,Z 318.852,A -85,B 0,C 180,E1 -13599.361,E2 -13599.361} C_VEL
LIN {X 0,Y 351.402,Z 319.211,A -85,B 0,C 180,E1 -13600.901,E2 -13600.901} C_VEL
LIN {X 0,Y 348.983,Z 319.509,A -85,B 0,C 180,E1 -13602.146,E2 -13602.146} C_VEL
LIN {X 0,Y 347.956,Z 319.638,A -85,B 0,C 180,E1 -13603.11,E2 -13603.11} C_VEL
LIN {X 0,Y 347.877,Z 319.647,A -85,B 0,C 180,E1 -13603.437,E2 -13603.437} C_VEL
LIN {X 0,Y 347.841,Z 319.656,A -85,B 0,C 180,E1 -13606.431,E2 -13606.431} C_VEL
LIN {X 0,Y 347.853,Z 319.647,A -85,B 0,C 180,E1 -13608.861,E2 -13608.861} C_VEL
LIN {X 0,Y 347.77,Z 319.659,A -85,B 0,C 180,E1 -13612.58,E2 -13612.58} C_VEL
LIN {X 0,Y 347.814,Z 319.66,A -85,B 0,C 180,E1 -13615.108,E2 -13615.108} C_VEL
LIN {X 0,Y 347.81,Z 319.649,A -85,B 0,C 180,E1 -13617.694,E2 -13617.694} C_VEL
LIN {X 0,Y 347.751,Z 319.663,A -85,B 0,C 180,E1 -13620.348,E2 -13620.348} C_VEL
LIN {X 0,Y 347.75,Z 319.652,A -85,B 0,C 180,E1 -13624.044,E2 -13624.044} C_VEL
LIN {X 0,Y 347.764,Z 319.664,A -85,B 0,C 180,E1 -13627.321,E2 -13627.321} C_VEL
LIN {X 0,Y 347.734,Z 319.657,A -85,B 0,C 180,E1 -13630.297,E2 -13630.297} C_VEL
LIN {X 0,Y 347.729,Z 319.659,A -85,B 0,C 180,E1 -13633.408,E2 -13633.408} C_VEL
LIN {X 0,Y 347.727,Z 319.67,A -85,B 0,C 180,E1 -13636.686,E2 -13636.686} C_VEL
LIN {X 0,Y 347.729,Z 319.647,A -85,B 0,C 180,E1 -13640.177,E2 -13640.177} C_VEL
LIN {X 0,Y 347.759,Z 319.653,A -85,B 0,C 180,E1 -13642.679,E2 -13642.679} C_VEL
LIN {X 0,Y 347.75,Z 319.664,A -85,B 0,C 180,E1 -13645.956,E2 -13645.956} C_VEL
LIN {X 0,Y 347.743,Z 319.643,A -85,B 0,C 180,E1 -13649.651,E2 -13649.651} C_VEL
LIN {X 0,Y 347.772,Z 319.653,A -85,B 0,C 180,E1 -13653.603,E2 -13653.603} C_VEL
LIN {X 0,Y 347.777,Z 319.665,A -85,B 0,C 180,E1 -13656.161,E2 -13656.161} C_VEL
LIN {X 0,Y 347.802,Z 319.645,A -85,B 0,C 180,E1 -13659.908,E2 -13659.908} C_VEL
LIN {X 0,Y 347.834,Z 319.639,A -85,B 0,C 180,E1 -13663.568,E2 -13663.568} C_VEL
LIN {X 0,Y 347.892,Z 319.649,A -85,B 0,C 180,E1 -13667.16,E2 -13667.16} C_VEL
LIN {X 0,Y 347.937,Z 319.632,A -85,B 0,C 180,E1 -13670.7,E2 -13670.7} C_VEL
LIN {X 0,Y 348.042,Z 319.602,A -85,B 0,C 180,E1 -13674.205,E2 -13674.205} C_VEL
LIN {X 0,Y 348.191,Z 319.604,A -85,B 0,C 180,E1 -13677.686,E2 -13677.686} C_VEL
LIN {X 0,Y 348.142,Z 319.61,A -85,B 0,C 180,E1 -13681.156,E2 -13681.156} C_VEL
LIN {X 0,Y 348.189,Z 319.602,A -85,B 0,C 180,E1 -13682.313,E2 -13682.313} C_VEL
LIN {X 0,Y 348.074,Z 319.611,A -85,B 0,C 180,E1 -13686.958,E2 -13686.958} C_VEL
LIN {X 0,Y 347.897,Z 319.646,A -85,B 0,C 180,E1 -13690.475,E2 -13690.475} C_VEL
LIN {X 0,Y 347.881,Z 319.629,A -85,B 0,C 180,E1 -13694.137,E2 -13694.137} C_VEL
LIN {X 0,Y 347.796,Z 319.661,A -85,B 0,C 180,E1 -13698.242,E2 -13698.242} C_VEL
LIN {X 0,Y 347.765,Z 319.661,A -85,B 0,C 180,E1 -13701.624,E2 -13701.624} C_VEL
LIN {X 0,Y 347.767,Z 319.656,A -85,B 0,C 180,E1 -13705.112,E2 -13705.112} C_VEL
LIN {X 0,Y 347.744,Z 319.665,A -85,B 0,C 180,E1 -13709.015,E2 -13709.015} C_VEL
LIN {X 0,Y 347.738,Z 319.66,A -85,B 0,C 180,E1 -13711.913,E2 -13711.913} C_VEL
LIN {X 0,Y 347.786,Z 319.657,A -85,B 0,C 180,E1 -13715.875,E2 -13715.875} C_VEL
LIN {X 0,Y 347.73,Z 319.665,A -85,B 0,C 180,E1 -13718.795,E2 -13718.795} C_VEL
LIN {X 0,Y 347.738,Z 319.664,A -85,B 0,C 180,E1 -13721.832,E2 -13721.832} C_VEL
LIN {X 0,Y 347.698,Z 319.671,A -85,B 0,C 180,E1 -13725.027,E2 -13725.027} C_VEL
LIN {X 0,Y 347.736,Z 319.672,A -85,B 0,C 180,E1 -13728.399,E2 -13728.399} C_VEL
LIN {X 0,Y 347.76,Z 319.663,A -85,B 0,C 180,E1 -13732.014,E2 -13732.014} C_VEL
LIN {X 0,Y 347.741,Z 319.664,A -85,B 0,C 180,E1 -13735.536,E2 -13735.536} C_VEL
LIN {X 0,Y 347.743,Z 319.669,A -85,B 0,C 180,E1 -13738.3,E2 -13738.3} C_VEL
LIN {X 0,Y 347.793,Z 319.844,A -85,B 0,C 180,E1 -13740.545,E2 -13740.545} C_VEL
LIN {X 0,Y 350.16,Z 331.112,A -85,B 0,C 180,E1 -13743.796,E2 -13743.796} C_VEL
LIN {X 0,Y 351.403,Z 338.394,A -85,B 0,C 180,E1 -13745.795,E2 -13745.795} C_VEL
LIN {X 0,Y 350.899,Z 344.495,A -85,B 0,C 180,E1 -13747.296,E2 -13747.296} C_VEL
LIN {X 0,Y 351.543,Z 348.489,A -85,B 0,C 180,E1 -13747.489,E2 -13747.489} C_VEL
LIN {X 0,Y 356.342,Z 377.504,A -85,B 0,C 180,E1 -13748.408,E2 -13748.408} C_VEL
LIN {X 0,Y 354.976,Z 451.307,A -85,B 0,C 180,E1 -13749.955,E2 -13749.955} C_VEL
LIN {X 0,Y 354.643,Z 460.908,A -85,B 0,C 180,E1 -13750.275,E2 -13750.275} C_VEL
LIN {X 0,Y 353.943,Z 470.755,A -85,B 0,C 180,E1 -13750.724,E2 -13750.724} C_VEL
LIN {X 0,Y 353.209,Z 481.984,A -85,B 0,C 180,E1 -13751.436,E2 -13751.436} C_VEL
LIN {X 0,Y 352.194,Z 492.44,A -85,B 0,C 180,E1 -13752.283,E2 -13752.283} C_VEL
LIN {X 0,Y 351.371,Z 501.042,A -85,B 0,C 180,E1 -13753.14,E2 -13753.14} C_VEL
LIN {X 0,Y 350.357,Z 510.803,A -85,B 0,C 180,E1 -13754.334,E2 -13754.334} C_VEL
LIN {X 0,Y 349.515,Z 518.404,A -85,B 0,C 180,E1 -13755.443,E2 -13755.443} C_VEL
LIN {X 0,Y 348.616,Z 526.614,A -85,B 0,C 180,E1 -13756.891,E2 -13756.891} C_VEL
LIN {X 0,Y 347.767,Z 533.442,A -85,B 0,C 180,E1 -13758.341,E2 -13758.341} C_VEL
LIN {X 0,Y 347.321,Z 538.148,A -85,B 0,C 180,E1 -13759.507,E2 -13759.507} C_VEL
LIN {X 0,Y 346.765,Z 543.905,A -85,B 0,C 180,E1 -13761.257,E2 -13761.257} C_VEL
LIN {X 0,Y 346.416,Z 548.43,A -85,B 0,C 180,E1 -13763.008,E2 -13763.008} C_VEL
LIN {X 0,Y 346.165,Z 552.687,A -85,B 0,C 180,E1 -13765.342,E2 -13765.342} C_VEL
LIN {X 0,Y 346.12,Z 554.291,A -85,B 0,C 180,E1 -13766.508,E2 -13766.508} C_VEL
LIN {X 0,Y 346.046,Z 555.991,A -85,B 0,C 180,E1 -13768.836,E2 -13768.836} C_VEL
LIN {X 0,Y 346.072,Z 556.308,A -85,B 0,C 180,E1 -13770,E2 -13770} C_VEL
LIN {X 0,Y 346.044,Z 555.666,A -85,B 0,C 180,E1 -13772.328,E2 -13772.328} C_VEL
LIN {X 0,Y 346.126,Z 554.691,A -85,B 0,C 180,E1 -13773.492,E2 -13773.492} C_VEL
LIN {X 0,Y 346.265,Z 551.66,A -85,B 0,C 180,E1 -13775.824,E2 -13775.824} C_VEL
LIN {X 0,Y 346.523,Z 548.171,A -85,B 0,C 180,E1 -13777.575,E2 -13777.575} C_VEL
LIN {X 0,Y 346.967,Z 543.598,A -85,B 0,C 180,E1 -13779.325,E2 -13779.325} C_VEL
LIN {X 0,Y 347.805,Z 536.624,A -85,B 0,C 180,E1 -13781.362,E2 -13781.362} C_VEL
LIN {X 0,Y 348.564,Z 530.51,A -85,B 0,C 180,E1 -13782.814,E2 -13782.814} C_VEL
LIN {X 0,Y 349.57,Z 523.145,A -85,B 0,C 180,E1 -13784.258,E2 -13784.258} C_VEL
LIN {X 0,Y 350.459,Z 515.255,A -85,B 0,C 180,E1 -13785.553,E2 -13785.553} C_VEL
LIN {X 0,Y 351.628,Z 505.599,A -85,B 0,C 180,E1 -13786.847,E2 -13786.847} C_VEL
LIN {X 0,Y 352.662,Z 496.584,A -85,B 0,C 180,E1 -13787.842,E2 -13787.842} C_VEL
LIN {X 0,Y 353.687,Z 487.242,A -85,B 0,C 180,E1 -13788.688,E2 -13788.688} C_VEL
LIN {X 0,Y 354.634,Z 476.473,A -85,B 0,C 180,E1 -13789.462,E2 -13789.462} C_VEL
LIN {X 0,Y 355.532,Z 464.754,A -85,B 0,C 180,E1 -13790.088,E2 -13790.088} C_VEL
LIN {X 0,Y 356.124,Z 454.928,A -85,B 0,C 180,E1 -13790.467,E2 -13790.467} C_VEL
LIN {X 0,Y 356.582,Z 437.143,A -85,B 0,C 180,E1 -13790.894,E2 -13790.894} C_VEL
LIN {X 0,Y 357.674,Z 377.258,A -85,B 0,C 180,E1 -13792.142,E2 -13792.142} C_VEL
LIN {X 0,Y 353.64,Z 354.327,A -85,B 0,C 180,E1 -13792.951,E2 -13792.951} C_VEL
LIN {X 0,Y 351.623,Z 344.334,A -85,B 0,C 180,E1 -13793.358,E2 -13793.358} C_VEL
LIN {X 0,Y 351.748,Z 341.927,A -85,B 0,C 180,E1 -13793.866,E2 -13793.866} C_VEL
LIN {X 0,Y 351.878,Z 339.464,A -85,B 0,C 180,E1 -13794.484,E2 -13794.484} C_VEL
LIN {X 0,Y 349.532,Z 327.51,A -85,B 0,C 180,E1 -13797.786,E2 -13797.786} C_VEL
LIN {X 0,Y 347.812,Z 319.759,A -85,B 0,C 180,E1 -13800.097,E2 -13800.097} C_VEL
LIN {X 0,Y 347.746,Z 319.663,A -85,B 0,C 180,E1 -13804.044,E2 -13804.044} C_VEL
LIN {X 0,Y 347.759,Z 319.662,A -85,B 0,C 180,E1 -13807.321,E2 -13807.321} C_VEL
LIN {X 0,Y 347.726,Z 319.659,A -85,B 0,C 180,E1 -13810.298,E2 -13810.298} C_VEL
LIN {X 0,Y 347.721,Z 319.67,A -85,B 0,C 180,E1 -13813.408,E2 -13813.408} C_VEL
LIN {X 0,Y 347.723,Z 319.669,A -85,B 0,C 180,E1 -13816.687,E2 -13816.687} C_VEL
LIN {X 0,Y 347.746,Z 319.667,A -85,B 0,C 180,E1 -13820.173,E2 -13820.173} C_VEL
LIN {X 0,Y 347.76,Z 319.665,A -85,B 0,C 180,E1 -13822.679,E2 -13822.679} C_VEL
LIN {X 0,Y 347.747,Z 319.665,A -85,B 0,C 180,E1 -13825.957,E2 -13825.957} C_VEL
LIN {X 0,Y 347.748,Z 319.663,A -85,B 0,C 180,E1 -13829.652,E2 -13829.652} C_VEL
LIN {X 0,Y 347.831,Z 319.653,A -85,B 0,C 180,E1 -13833.608,E2 -13833.608} C_VEL
LIN {X 0,Y 347.788,Z 319.659,A -85,B 0,C 180,E1 -13836.162,E2 -13836.162} C_VEL
LIN {X 0,Y 347.817,Z 319.656,A -85,B 0,C 180,E1 -13839.91,E2 -13839.91} C_VEL
LIN {X 0,Y 347.867,Z 319.645,A -85,B 0,C 180,E1 -13842.36,E2 -13842.36} C_VEL
LIN {X 0,Y 347.898,Z 319.639,A -85,B 0,C 180,E1 -13845.971,E2 -13845.971} C_VEL
LIN {X 0,Y 347.93,Z 319.646,A -85,B 0,C 180,E1 -13849.526,E2 -13849.526} C_VEL
LIN {X 0,Y 348.109,Z 319.62,A -85,B 0,C 180,E1 -13853.043,E2 -13853.043} C_VEL
LIN {X 0,Y 348.21,Z 319.607,A -85,B 0,C 180,E1 -13857.687,E2 -13857.687} C_VEL
LIN {X 0,Y 348.348,Z 319.587,A -85,B 0,C 180,E1 -13860,E2 -13860} C_VEL
LIN {X 0,Y 348.209,Z 319.609,A -85,B 0,C 180,E1 -13862.314,E2 -13862.314} C_VEL
LIN {X 0,Y 348.108,Z 319.625,A -85,B 0,C 180,E1 -13866.958,E2 -13866.958} C_VEL
LIN {X 0,Y 347.969,Z 319.636,A -85,B 0,C 180,E1 -13869.299,E2 -13869.299} C_VEL
LIN {X 0,Y 347.891,Z 319.643,A -85,B 0,C 180,E1 -13872.84,E2 -13872.84} C_VEL
LIN {X 0,Y 347.841,Z 319.653,A -85,B 0,C 180,E1 -13876.432,E2 -13876.432} C_VEL
LIN {X 0,Y 347.852,Z 319.65,A -85,B 0,C 180,E1 -13878.861,E2 -13878.861} C_VEL
LIN {X 0,Y 347.763,Z 319.667,A -85,B 0,C 180,E1 -13882.58,E2 -13882.58} C_VEL
LIN {X 0,Y 347.796,Z 319.662,A -85,B 0,C 180,E1 -13885.11,E2 -13885.11} C_VEL
LIN {X 0,Y 347.79,Z 319.649,A -85,B 0,C 180,E1 -13887.696,E2 -13887.696} C_VEL
LIN {X 0,Y 347.75,Z 319.665,A -85,B 0,C 180,E1 -13890.348,E2 -13890.348} C_VEL
LIN {X 0,Y 347.749,Z 319.661,A -85,B 0,C 180,E1 -13894.044,E2 -13894.044} C_VEL
LIN {X 0,Y 347.766,Z 319.668,A -85,B 0,C 180,E1 -13897.32,E2 -13897.32} C_VEL
LIN {X 0,Y 347.79,Z 319.742,A -85,B 0,C 180,E1 -13898.292,E2 -13898.292} C_VEL
LIN {X 0,Y 349.227,Z 325.86,A -85,B 0,C 180,E1 -13900.117,E2 -13900.117} C_VEL
LIN {X 0,Y 351.117,Z 335.2,A -85,B 0,C 180,E1 -13902.628,E2 -13902.628} C_VEL
LIN {X 0,Y 353.315,Z 341.65,A -85,B 0,C 180,E1 -13902.981,E2 -13902.981} C_VEL
LIN {X 0,Y 357.605,Z 362.824,A -85,B 0,C 180,E1 -13903.777,E2 -13903.777} C_VEL
LIN {X 0,Y 357.939,Z 367.274,A -85,B 0,C 180,E1 -13903.899,E2 -13903.899} C_VEL
LIN {X 0,Y 356.266,Z 441.493,A -85,B 0,C 180,E1 -13905.457,E2 -13905.457} C_VEL
LIN {X 0,Y 355.789,Z 451.887,A -85,B 0,C 180,E1 -13905.8,E2 -13905.8} C_VEL
LIN {X 0,Y 355.281,Z 461.763,A -85,B 0,C 180,E1 -13906.272,E2 -13906.272} C_VEL
LIN {X 0,Y 354.444,Z 472.279,A -85,B 0,C 180,E1 -13906.932,E2 -13906.932} C_VEL
LIN {X 0,Y 353.628,Z 481.685,A -85,B 0,C 180,E1 -13907.683,E2 -13907.683} C_VEL
LIN {X 0,Y 352.584,Z 491.701,A -85,B 0,C 180,E1 -13908.679,E2 -13908.679} C_VEL
LIN {X 0,Y 351.629,Z 499.776,A -85,B 0,C 180,E1 -13909.64,E2 -13909.64} C_VEL
LIN {X 0,Y 350.537,Z 508.142,A -85,B 0,C 180,E1 -13910.835,E2 -13910.835} C_VEL
LIN {X 0,Y 349.534,Z 515.911,A -85,B 0,C 180,E1 -13912.175,E2 -13912.175} C_VEL
LIN {X 0,Y 348.55,Z 523.444,A -85,B 0,C 180,E1 -13913.76,E2 -13913.76} C_VEL
LIN {X 0,Y 347.671,Z 530.222,A -85,B 0,C 180,E1 -13915.528,E2 -13915.528} C_VEL
LIN {X 0,Y 347.161,Z 534.503,A -85,B 0,C 180,E1 -13916.866,E2 -13916.866} C_VEL
LIN {X 0,Y 346.587,Z 539.585,A -85,B 0,C 180,E1 -13918.944,E2 -13918.944} C_VEL
LIN {X 0,Y 346.288,Z 542.875,A -85,B 0,C 180,E1 -13920.774,E2 -13920.774} C_VEL
LIN {X 0,Y 346.061,Z 544.732,A -85,B 0,C 180,E1 -13922.154,E2 -13922.154} C_VEL
LIN {X 0,Y 345.909,Z 545.803,A -85,B 0,C 180,E1 -13923.45,E2 -13923.45} C_VEL
LIN {X 0,Y 345.795,Z 546.643,A -85,B 0,C 180,E1 -13926.016,E2 -13926.016} C_VEL
LIN {X 0,Y 345.816,Z 546.285,A -85,B 0,C 180,E1 -13927.286,E2 -13927.286} C_VEL
LIN {X 0,Y 346.024,Z 544.255,A -85,B 0,C 180,E1 -13929.801,E2 -13929.801} C_VEL
LIN {X 0,Y 346.31,Z 541.467,A -85,B 0,C 180,E1 -13931.666,E2 -13931.666} C_VEL
LIN {X 0,Y 346.658,Z 537.57,A -85,B 0,C 180,E1 -13933.511,E2 -13933.511} C_VEL
LIN {X 0,Y 347.142,Z 532.457,A -85,B 0,C 180,E1 -13935.341,E2 -13935.341} C_VEL
LIN {X 0,Y 347.625,Z 527.966,A -85,B 0,C 180,E1 -13936.667,E2 -13936.667} C_VEL
LIN {X 0,Y 348.418,Z 520.832,A -85,B 0,C 180,E1 -13938.363,E2 -13938.363} C_VEL
LIN {X 0,Y 349.233,Z 513.749,A -85,B 0,C 180,E1 -13939.754,E2 -13939.754} C_VEL
LIN {X 0,Y 350.155,Z 505.818,A -85,B 0,C 180,E1 -13941.051,E2 -13941.051} C_VEL
LIN {X 0,Y 351.072,Z 497.129,A -85,B 0,C 180,E1 -13942.234,E2 -13942.234} C_VEL
LIN {X 0,Y 352.061,Z 487.936,A -85,B 0,C 180,E1 -13943.265,E2 -13943.265} C_VEL
LIN {X 0,Y 352.914,Z 478.436,A -85,B 0,C 180,E1 -13944.142,E2 -13944.142} C_VEL
LIN {X 0,Y 353.822,Z 466.746,A -85,B 0,C 180,E1 -13944.982,E2 -13944.982} C_VEL
LIN {X 0,Y 354.45,Z 455.453,A -85,B 0,C 180,E1 -13945.594,E2 -13945.594} C_VEL
LIN {X 0,Y 354.993,Z 445.049,A -85,B 0,C 180,E1 -13945.991,E2 -13945.991} C_VEL
LIN {X 0,Y 355.395,Z 428.499,A -85,B 0,C 180,E1 -13946.386,E2 -13946.386} C_VEL
LIN {X 0,Y 356.465,Z 363.804,A -85,B 0,C 180,E1 -13947.722,E2 -13947.722} C_VEL
LIN {X 0,Y 351.175,Z 336.478,A -85,B 0,C 180,E1 -13948.654,E2 -13948.654} C_VEL
LIN {X 0,Y 350.972,Z 335.319,A -85,B 0,C 180,E1 -13948.782,E2 -13948.782} C_VEL
LIN {X 0,Y 350.044,Z 329.032,A -85,B 0,C 180,E1 -13950.575,E2 -13950.575} C_VEL
LIN {X 0,Y 348.162,Z 320.378,A -85,B 0,C 180,E1 -13953.182,E2 -13953.182} C_VEL
LIN {X 0,Y 347.961,Z 319.639,A -85,B 0,C 180,E1 -13953.619,E2 -13953.619} C_VEL
LIN {X 0,Y 348.079,Z 319.628,A -85,B 0,C 180,E1 -13956.958,E2 -13956.958} C_VEL
LIN {X 0,Y 347.899,Z 319.648,A -85,B 0,C 180,E1 -13960.475,E2 -13960.475} C_VEL
LIN {X 0,Y 347.877,Z 319.647,A -85,B 0,C 180,E1 -13963.437,E2 -13963.437} C_VEL
LIN {X 0,Y 347.234,Z 319.732,A -85,B 0,C 180,E1 -13964.403,E2 -13964.403} C_VEL
LIN {X 0,Y 344.426,Z 320.084,A -85,B 0,C 180,E1 -13965.976,E2 -13965.976} C_VEL
LIN {X 0,Y 342.012,Z 320.382,A -85,B 0,C 180,E1 -13967.249,E2 -13967.249} C_VEL
LIN {X 0,Y 340.937,Z 320.513,A -85,B 0,C 180,E1 -13968.233,E2 -13968.233} C_VEL
LIN {X 0,Y 340.829,Z 320.522,A -85,B 0,C 180,E1 -13968.567,E2 -13968.567} C_VEL
LIN {X 0,Y 340.723,Z 320.542,A -85,B 0,C 180,E1 -13971.843,E2 -13971.843} C_VEL
LIN {X 0,Y 340.774,Z 320.534,A -85,B 0,C 180,E1 -13975.664,E2 -13975.664} C_VEL
LIN {X 0,Y 340.73,Z 320.53,A -85,B 0,C 180,E1 -13978.321,E2 -13978.321} C_VEL
LIN {X 0,Y 340.7,Z 320.546,A -85,B 0,C 180,E1 -13981.045,E2 -13981.045} C_VEL
LIN {X 0,Y 340.72,Z 320.53,A -85,B 0,C 180,E1 -13985.279,E2 -13985.279} C_VEL
LIN {X 0,Y 340.711,Z 320.542,A -85,B 0,C 180,E1 -13988.386,E2 -13988.386} C_VEL
LIN {X 0,Y 340.701,Z 320.528,A -85,B 0,C 180,E1 -13992.045,E2 -13992.045} C_VEL
LIN {X 0,Y 340.684,Z 320.544,A -85,B 0,C 180,E1 -13995.461,E2 -13995.461} C_VEL
LIN {X 0,Y 340.681,Z 320.535,A -85,B 0,C 180,E1 -13998.69,E2 -13998.69} C_VEL
LIN {X 0,Y 340.722,Z 320.528,A -85,B 0,C 180,E1 -14001.771,E2 -14001.771} C_VEL
LIN {X 0,Y 340.725,Z 320.542,A -85,B 0,C 180,E1 -14005.595,E2 -14005.595} C_VEL
LIN {X 0,Y 340.696,Z 320.531,A -85,B 0,C 180,E1 -14008.955,E2 -14008.955} C_VEL
LIN {X 0,Y 340.73,Z 320.528,A -85,B 0,C 180,E1 -14013.013,E2 -14013.013} C_VEL
LIN {X 0,Y 340.758,Z 320.535,A -85,B 0,C 180,E1 -14015.638,E2 -14015.638} C_VEL
LIN {X 0,Y 340.734,Z 320.525,A -85,B 0,C 180,E1 -14019.473,E2 -14019.473} C_VEL
LIN {X 0,Y 340.794,Z 320.497,A -85,B 0,C 180,E1 -14021.981,E2 -14021.981} C_VEL
LIN {X 0,Y 340.872,Z 320.519,A -85,B 0,C 180,E1 -14025.705,E2 -14025.705} C_VEL
LIN {X 0,Y 340.85,Z 320.525,A -85,B 0,C 180,E1 -14029.305,E2 -14029.305} C_VEL
LIN {X 0,Y 341.003,Z 320.478,A -85,B 0,C 180,E1 -14032.896,E2 -14032.896} C_VEL
LIN {X 0,Y 340.817,Z 320.507,A -85,B 0,C 180,E1 -14035.268,E2 -14035.268} C_VEL
LIN {X 0,Y 341.128,Z 320.484,A -85,B 0,C 180,E1 -14037.638,E2 -14037.638} C_VEL
LIN {X 0,Y 341.111,Z 320.486,A -85,B 0,C 180,E1 -14041.18,E2 -14041.18} C_VEL
LIN {X 0,Y 341.127,Z 320.481,A -85,B 0,C 180,E1 -14042.361,E2 -14042.361} C_VEL
LIN {X 0,Y 341.043,Z 320.489,A -85,B 0,C 180,E1 -14047.102,E2 -14047.102} C_VEL
LIN {X 0,Y 340.849,Z 320.525,A -85,B 0,C 180,E1 -14050.694,E2 -14050.694} C_VEL
LIN {X 0,Y 340.819,Z 320.507,A -85,B 0,C 180,E1 -14054.326,E2 -14054.326} C_VEL
LIN {X 0,Y 340.758,Z 320.538,A -85,B 0,C 180,E1 -14058.425,E2 -14058.425} C_VEL
LIN {X 0,Y 340.719,Z 320.54,A -85,B 0,C 180,E1 -14061.841,E2 -14061.841} C_VEL
LIN {X 0,Y 340.715,Z 320.535,A -85,B 0,C 180,E1 -14065.669,E2 -14065.669} C_VEL
LIN {X 0,Y 340.705,Z 320.536,A -85,B 0,C 180,E1 -14069.674,E2 -14069.674} C_VEL
LIN {X 0,Y 340.686,Z 320.538,A -85,B 0,C 180,E1 -14072.435,E2 -14072.435} C_VEL
LIN {X 0,Y 340.717,Z 320.546,A -85,B 0,C 180,E1 -14075.279,E2 -14075.279} C_VEL
LIN {X 0,Y 340.693,Z 320.543,A -85,B 0,C 180,E1 -14078.382,E2 -14078.382} C_VEL
LIN {X 0,Y 340.689,Z 320.541,A -85,B 0,C 180,E1 -14082.043,E2 -14082.043} C_VEL
LIN {X 0,Y 340.648,Z 320.55,A -85,B 0,C 180,E1 -14086.227,E2 -14086.227} C_VEL
LIN {X 0,Y 340.666,Z 320.549,A -85,B 0,C 180,E1 -14088.687,E2 -14088.687} C_VEL
LIN {X 0,Y 340.717,Z 320.541,A -85,B 0,C 180,E1 -14091.77,E2 -14091.77} C_VEL
LIN {X 0,Y 340.72,Z 320.538,A -85,B 0,C 180,E1 -14095.595,E2 -14095.595} C_VEL
LIN {X 0,Y 340.691,Z 320.543,A -85,B 0,C 180,E1 -14098.954,E2 -14098.954} C_VEL
LIN {X 0,Y 340.729,Z 320.663,A -85,B 0,C 180,E1 -14100.153,E2 -14100.153} C_VEL
LIN {X 0,Y 343.343,Z 333.109,A -85,B 0,C 180,E1 -14103.838,E2 -14103.838} C_VEL
LIN {X 0,Y 344.429,Z 339.365,A -85,B 0,C 180,E1 -14105.594,E2 -14105.594} C_VEL
LIN {X 0,Y 344.051,Z 344.563,A -85,B 0,C 180,E1 -14106.878,E2 -14106.878} C_VEL
LIN {X 0,Y 345.75,Z 354.116,A -85,B 0,C 180,E1 -14107.249,E2 -14107.249} C_VEL
LIN {X 0,Y 349.613,Z 377.32,A -85,B 0,C 180,E1 -14108.003,E2 -14108.003} C_VEL
LIN {X 0,Y 348.349,Z 448.684,A -85,B 0,C 180,E1 -14109.518,E2 -14109.518} C_VEL
LIN {X 0,Y 347.909,Z 459.997,A -85,B 0,C 180,E1 -14109.876,E2 -14109.876} C_VEL
LIN {X 0,Y 347.13,Z 471.275,A -85,B 0,C 180,E1 -14110.408,E2 -14110.408} C_VEL
LIN {X 0,Y 346.471,Z 481.428,A -85,B 0,C 180,E1 -14111.061,E2 -14111.061} C_VEL
LIN {X 0,Y 345.415,Z 491.977,A -85,B 0,C 180,E1 -14111.923,E2 -14111.923} C_VEL
LIN {X 0,Y 344.413,Z 501.885,A -85,B 0,C 180,E1 -14112.942,E2 -14112.942} C_VEL
LIN {X 0,Y 343.531,Z 510.148,A -85,B 0,C 180,E1 -14113.967,E2 -14113.967} C_VEL
LIN {X 0,Y 342.627,Z 518.109,A -85,B 0,C 180,E1 -14115.143,E2 -14115.143} C_VEL
LIN {X 0,Y 341.678,Z 526.356,A -85,B 0,C 180,E1 -14116.62,E2 -14116.62} C_VEL
LIN {X 0,Y 340.784,Z 533.215,A -85,B 0,C 180,E1 -14118.098,E2 -14118.098} C_VEL
LIN {X 0,Y 340.329,Z 537.932,A -85,B 0,C 180,E1 -14119.289,E2 -14119.289} C_VEL
LIN {X 0,Y 339.725,Z 543.72,A -85,B 0,C 180,E1 -14121.074,E2 -14121.074} C_VEL
LIN {X 0,Y 339.346,Z 548.268,A -85,B 0,C 180,E1 -14122.862,E2 -14122.862} C_VEL
LIN {X 0,Y 339.07,Z 552.548,A -85,B 0,C 180,E1 -14125.244,E2 -14125.244} C_VEL
LIN {X 0,Y 339.046,Z 554.16,A -85,B 0,C 180,E1 -14126.435,E2 -14126.435} C_VEL
LIN {X 0,Y 338.952,Z 555.884,A -85,B 0,C 180,E1 -14128.812,E2 -14128.812} C_VEL
LIN {X 0,Y 338.975,Z 556.201,A -85,B 0,C 180,E1 -14130,E2 -14130} C_VEL
LIN {X 0,Y 338.961,Z 555.59,A -85,B 0,C 180,E1 -14132.377,E2 -14132.377} C_VEL
LIN {X 0,Y 339.054,Z 554.615,A -85,B 0,C 180,E1 -14133.565,E2 -14133.565} C_VEL
LIN {X 0,Y 339.203,Z 551.509,A -85,B 0,C 180,E1 -14136.006,E2 -14136.006} C_VEL
LIN {X 0,Y 339.484,Z 548.14,A -85,B 0,C 180,E1 -14137.733,E2 -14137.733} C_VEL
LIN {X 0,Y 339.944,Z 543.586,A -85,B 0,C 180,E1 -14139.52,E2 -14139.52} C_VEL
LIN {X 0,Y 340.792,Z 536.646,A -85,B 0,C 180,E1 -14141.599,E2 -14141.599} C_VEL
LIN {X 0,Y 341.65,Z 530.557,A -85,B 0,C 180,E1 -14143.078,E2 -14143.078} C_VEL
LIN {X 0,Y 342.688,Z 523.219,A -85,B 0,C 180,E1 -14144.55,E2 -14144.55} C_VEL
LIN {X 0,Y 343.706,Z 514.729,A -85,B 0,C 180,E1 -14145.961,E2 -14145.961} C_VEL
LIN {X 0,Y 344.834,Z 505.749,A -85,B 0,C 180,E1 -14147.189,E2 -14147.189} C_VEL
LIN {X 0,Y 345.929,Z 496.788,A -85,B 0,C 180,E1 -14148.202,E2 -14148.202} C_VEL
LIN {X 0,Y 346.993,Z 487.519,A -85,B 0,C 180,E1 -14149.062,E2 -14149.062} C_VEL
LIN {X 0,Y 347.973,Z 476.86,A -85,B 0,C 180,E1 -14149.85,E2 -14149.85} C_VEL
LIN {X 0,Y 348.9,Z 465.34,A -85,B 0,C 180,E1 -14150.487,E2 -14150.487} C_VEL
LIN {X 0,Y 349.559,Z 454.644,A -85,B 0,C 180,E1 -14150.908,E2 -14150.908} C_VEL
LIN {X 0,Y 350.073,Z 435.363,A -85,B 0,C 180,E1 -14151.374,E2 -14151.374} C_VEL
LIN {X 0,Y 351.189,Z 378.389,A -85,B 0,C 180,E1 -14152.584,E2 -14152.584} C_VEL
LIN {X 0,Y 347.364,Z 356.323,A -85,B 0,C 180,E1 -14153.381,E2 -14153.381} C_VEL
LIN {X 0,Y 344.882,Z 344.218,A -85,B 0,C 180,E1 -14153.893,E2 -14153.893} C_VEL
LIN {X 0,Y 345.007,Z 341.997,A -85,B 0,C 180,E1 -14154.362,E2 -14154.362} C_VEL
LIN {X 0,Y 343.883,Z 335.106,A -85,B 0,C 180,E1 -14156.265,E2 -14156.265} C_VEL
LIN {X 0,Y 341.674,Z 324.813,A -85,B 0,C 180,E1 -14159.243,E2 -14159.243} C_VEL
LIN {X 0,Y 340.732,Z 320.578,A -85,B 0,C 180,E1 -14160.61,E2 -14160.61} C_VEL
LIN {X 0,Y 340.721,Z 320.539,A -85,B 0,C 180,E1 -14164.405,E2 -14164.405} C_VEL
LIN {X 0,Y 340.708,Z 320.546,A -85,B 0,C 180,E1 -14168.386,E2 -14168.386} C_VEL
LIN {X 0,Y 340.694,Z 320.546,A -85,B 0,C 180,E1 -14172.045,E2 -14172.045} C_VEL
LIN {X 0,Y 340.65,Z 320.55,A -85,B 0,C 180,E1 -14176.227,E2 -14176.227} C_VEL
LIN {X 0,Y 340.687,Z 320.55,A -85,B 0,C 180,E1 -14179.753,E2 -14179.753} C_VEL
LIN {X 0,Y 340.704,Z 320.545,A -85,B 0,C 180,E1 -14183.259,E2 -14183.259} C_VEL
LIN {X 0,Y 340.693,Z 320.546,A -85,B 0,C 180,E1 -14186.154,E2 -14186.154} C_VEL
LIN {X 0,Y 340.741,Z 320.542,A -85,B 0,C 180,E1 -14190.33,E2 -14190.33} C_VEL
LIN {X 0,Y 340.803,Z 320.527,A -85,B 0,C 180,E1 -14193.02,E2 -14193.02} C_VEL
LIN {X 0,Y 340.756,Z 320.535,A -85,B 0,C 180,E1 -14195.639,E2 -14195.639} C_VEL
LIN {X 0,Y 340.749,Z 320.539,A -85,B 0,C 180,E1 -14199.475,E2 -14199.475} C_VEL
LIN {X 0,Y 340.858,Z 320.518,A -85,B 0,C 180,E1 -14201.985,E2 -14201.985} C_VEL
LIN {X 0,Y 340.87,Z 320.516,A -85,B 0,C 180,E1 -14205.705,E2 -14205.705} C_VEL
LIN {X 0,Y 340.872,Z 320.524,A -85,B 0,C 180,E1 -14209.307,E2 -14209.307} C_VEL
LIN {X 0,Y 341.079,Z 320.496,A -85,B 0,C 180,E1 -14212.899,E2 -14212.899} C_VEL
LIN {X 0,Y 341.171,Z 320.484,A -85,B 0,C 180,E1 -14217.639,E2 -14217.639} C_VEL
LIN {X 0,Y 341.298,Z 320.465,A -85,B 0,C 180,E1 -14220,E2 -14220} C_VEL
LIN {X 0,Y 341.171,Z 320.486,A -85,B 0,C 180,E1 -14222.361,E2 -14222.361} C_VEL
LIN {X 0,Y 341.078,Z 320.501,A -85,B 0,C 180,E1 -14227.102,E2 -14227.102} C_VEL
LIN {X 0,Y 340.873,Z 320.523,A -85,B 0,C 180,E1 -14230.694,E2 -14230.694} C_VEL
LIN {X 0,Y 340.864,Z 320.524,A -85,B 0,C 180,E1 -14234.325,E2 -14234.325} C_VEL
LIN {X 0,Y 340.838,Z 320.525,A -85,B 0,C 180,E1 -14238.467,E2 -14238.467} C_VEL
LIN {X 0,Y 340.719,Z 320.542,A -85,B 0,C 180,E1 -14241.842,E2 -14241.842} C_VEL
LIN {X 0,Y 340.753,Z 320.539,A -85,B 0,C 180,E1 -14245.666,E2 -14245.666} C_VEL
LIN {X 0,Y 340.719,Z 320.533,A -85,B 0,C 180,E1 -14248.322,E2 -14248.322} C_VEL
LIN {X 0,Y 340.698,Z 320.539,A -85,B 0,C 180,E1 -14251.045,E2 -14251.045} C_VEL
LIN {X 0,Y 340.719,Z 320.547,A -85,B 0,C 180,E1 -14255.279,E2 -14255.279} C_VEL
LIN {X 0,Y 340.745,Z 320.667,A -85,B 0,C 180,E1 -14257.851,E2 -14257.851} C_VEL
LIN {X 0,Y 343.125,Z 331.146,A -85,B 0,C 180,E1 -14260.953,E2 -14260.953} C_VEL
LIN {X 0,Y 343.948,Z 335.302,A -85,B 0,C 180,E1 -14262.054,E2 -14262.054} C_VEL
LIN {X 0,Y 346.974,Z 343.284,A -85,B 0,C 180,E1 -14262.53,E2 -14262.53} C_VEL
LIN {X 0,Y 351.33,Z 365.035,A -85,B 0,C 180,E1 -14263.365,E2 -14263.365} C_VEL
LIN {X 0,Y 351.195,Z 380.36,A -85,B 0,C 180,E1 -14263.704,E2 -14263.704} C_VEL
LIN {X 0,Y 349.678,Z 442.039,A -85,B 0,C 180,E1 -14265.03,E2 -14265.03} C_VEL
LIN {X 0,Y 349.278,Z 451.139,A -85,B 0,C 180,E1 -14265.332,E2 -14265.332} C_VEL
LIN {X 0,Y 348.689,Z 461.776,A -85,B 0,C 180,E1 -14265.843,E2 -14265.843} C_VEL
LIN {X 0,Y 347.821,Z 472.207,A -85,B 0,C 180,E1 -14266.508,E2 -14266.508} C_VEL
LIN {X 0,Y 346.975,Z 481.621,A -85,B 0,C 180,E1 -14267.27,E2 -14267.27} C_VEL
LIN {X 0,Y 345.827,Z 492.096,A -85,B 0,C 180,E1 -14268.334,E2 -14268.334} C_VEL
LIN {X 0,Y 344.677,Z 501.18,A -85,B 0,C 180,E1 -14269.463,E2 -14269.463} C_VEL
LIN {X 0,Y 343.58,Z 509.123,A -85,B 0,C 180,E1 -14270.646,E2 -14270.646} C_VEL
LIN {X 0,Y 342.561,Z 516.75,A -85,B 0,C 180,E1 -14272.013,E2 -14272.013} C_VEL
LIN {X 0,Y 341.707,Z 523.18,A -85,B 0,C 180,E1 -14273.384,E2 -14273.384} C_VEL
LIN {X 0,Y 340.717,Z 530.206,A -85,B 0,C 180,E1 -14275.242,E2 -14275.242} C_VEL
LIN {X 0,Y 340.105,Z 534.995,A -85,B 0,C 180,E1 -14276.797,E2 -14276.797} C_VEL
LIN {X 0,Y 339.521,Z 539.826,A -85,B 0,C 180,E1 -14278.836,E2 -14278.836} C_VEL
LIN {X 0,Y 339.266,Z 542.749,A -85,B 0,C 180,E1 -14280.464,E2 -14280.464} C_VEL
LIN {X 0,Y 339.046,Z 544.189,A -85,B 0,C 180,E1 -14281.526,E2 -14281.526} C_VEL
LIN {X 0,Y 338.833,Z 545.702,A -85,B 0,C 180,E1 -14283.113,E2 -14283.113} C_VEL
LIN {X 0,Y 338.739,Z 546.381,A -85,B 0,C 180,E1 -14284.17,E2 -14284.17} C_VEL
LIN {X 0,Y 338.709,Z 546.759,A -85,B 0,C 180,E1 -14285.92,E2 -14285.92} C_VEL
LIN {X 0,Y 338.746,Z 545.956,A -85,B 0,C 180,E1 -14288.072,E2 -14288.072} C_VEL
LIN {X 0,Y 338.901,Z 544.905,A -85,B 0,C 180,E1 -14289.357,E2 -14289.357} C_VEL
LIN {X 0,Y 339.152,Z 542.414,A -85,B 0,C 180,E1 -14291.265,E2 -14291.265} C_VEL
LIN {X 0,Y 339.474,Z 538.838,A -85,B 0,C 180,E1 -14293.152,E2 -14293.152} C_VEL
LIN {X 0,Y 339.954,Z 534.076,A -85,B 0,C 180,E1 -14295.024,E2 -14295.024} C_VEL
LIN {X 0,Y 340.612,Z 527.958,A -85,B 0,C 180,E1 -14296.881,E2 -14296.881} C_VEL
LIN {X 0,Y 341.35,Z 521.722,A -85,B 0,C 180,E1 -14298.42,E2 -14298.42} C_VEL
LIN {X 0,Y 342.393,Z 512.998,A -85,B 0,C 180,E1 -14300.149,E2 -14300.149} C_VEL
LIN {X 0,Y 343.353,Z 504.928,A -85,B 0,C 180,E1 -14301.466,E2 -14301.466} C_VEL
LIN {X 0,Y 344.368,Z 496.006,A -85,B 0,C 180,E1 -14302.672,E2 -14302.672} C_VEL
LIN {X 0,Y 345.314,Z 486.608,A -85,B 0,C 180,E1 -14303.72,E2 -14303.72} C_VEL
LIN {X 0,Y 346.223,Z 476.851,A -85,B 0,C 180,E1 -14304.605,E2 -14304.605} C_VEL
LIN {X 0,Y 347.101,Z 466.39,A -85,B 0,C 180,E1 -14305.355,E2 -14305.355} C_VEL
LIN {X 0,Y 347.695,Z 455.735,A -85,B 0,C 180,E1 -14305.943,E2 -14305.943} C_VEL
LIN {X 0,Y 348.256,Z 445.432,A -85,B 0,C 180,E1 -14306.348,E2 -14306.348} C_VEL
LIN {X 0,Y 348.675,Z 429.358,A -85,B 0,C 180,E1 -14306.742,E2 -14306.742} C_VEL
LIN {X 0,Y 349.791,Z 364.726,A -85,B 0,C 180,E1 -14308.104,E2 -14308.104} C_VEL
LIN {X 0,Y 344.707,Z 338.39,A -85,B 0,C 180,E1 -14309.013,E2 -14309.013} C_VEL
LIN {X 0,Y 343.913,Z 335.643,A -85,B 0,C 180,E1 -14309.179,E2 -14309.179} C_VEL
LIN {X 0,Y 342.682,Z 328.836,A -85,B 0,C 180,E1 -14311.175,E2 -14311.175} C_VEL
LIN {X 0,Y 341.55,Z 323.044,A -85,B 0,C 180,E1 -14312.949,E2 -14312.949} C_VEL
LIN {X 0,Y 340.873,Z 320.548,A -85,B 0,C 180,E1 -14313.842,E2 -14313.842} C_VEL
LIN {X 0,Y 341.047,Z 320.505,A -85,B 0,C 180,E1 -14317.103,E2 -14317.103} C_VEL
LIN {X 0,Y 340.85,Z 320.527,A -85,B 0,C 180,E1 -14320.695,E2 -14320.695} C_VEL
LIN {X 0,Y 340.865,Z 320.523,A -85,B 0,C 180,E1 -14324.325,E2 -14324.325} C_VEL
LIN {X 0,Y 340.829,Z 320.522,A -85,B 0,C 180,E1 -14328.567,E2 -14328.567} C_VEL
LIN {X 0,Y 340.099,Z 320.613,A -85,B 0,C 180,E1 -14329.552,E2 -14329.552} C_VEL
LIN {X 0,Y 337.201,Z 320.98,A -85,B 0,C 180,E1 -14331.155,E2 -14331.155} C_VEL
LIN {X 0,Y 334.783,Z 321.277,A -85,B 0,C 180,E1 -14332.453,E2 -14332.453} C_VEL
LIN {X 0,Y 333.752,Z 321.402,A -85,B 0,C 180,E1 -14333.458,E2 -14333.458} C_VEL
LIN {X 0,Y 333.67,Z 321.412,A -85,B 0,C 180,E1 -14333.799,E2 -14333.799} C_VEL
LIN {X 0,Y 333.741,Z 321.402,A -85,B 0,C 180,E1 -14337.599,E2 -14337.599} C_VEL
LIN {X 0,Y 333.692,Z 321.415,A -85,B 0,C 180,E1 -14340.363,E2 -14340.363} C_VEL
LIN {X 0,Y 333.676,Z 321.404,A -85,B 0,C 180,E1 -14344.659,E2 -14344.659} C_VEL
LIN {X 0,Y 333.654,Z 321.425,A -85,B 0,C 180,E1 -14347.651,E2 -14347.651} C_VEL
LIN {X 0,Y 333.648,Z 321.408,A -85,B 0,C 180,E1 -14350.767,E2 -14350.767} C_VEL
LIN {X 0,Y 333.628,Z 321.421,A -85,B 0,C 180,E1 -14354.256,E2 -14354.256} C_VEL
LIN {X 0,Y 333.642,Z 321.418,A -85,B 0,C 180,E1 -14357.618,E2 -14357.618} C_VEL
LIN {X 0,Y 333.641,Z 321.403,A -85,B 0,C 180,E1 -14361.205,E2 -14361.205} C_VEL
LIN {X 0,Y 333.677,Z 321.417,A -85,B 0,C 180,E1 -14363.861,E2 -14363.861} C_VEL
LIN {X 0,Y 333.645,Z 321.418,A -85,B 0,C 180,E1 -14367.413,E2 -14367.413} C_VEL
LIN {X 0,Y 333.657,Z 321.39,A -85,B 0,C 180,E1 -14371.023,E2 -14371.023} C_VEL
LIN {X 0,Y 333.717,Z 321.411,A -85,B 0,C 180,E1 -14375.09,E2 -14375.09} C_VEL
LIN {X 0,Y 333.673,Z 321.407,A -85,B 0,C 180,E1 -14379.018,E2 -14379.018} C_VEL
LIN {X 0,Y 333.743,Z 321.375,A -85,B 0,C 180,E1 -14381.586,E2 -14381.586} C_VEL
LIN {X 0,Y 333.811,Z 321.4,A -85,B 0,C 180,E1 -14385.577,E2 -14385.577} C_VEL
LIN {X 0,Y 333.819,Z 321.401,A -85,B 0,C 180,E1 -14389.077,E2 -14389.077} C_VEL
LIN {X 0,Y 333.958,Z 321.355,A -85,B 0,C 180,E1 -14392.746,E2 -14392.746} C_VEL
LIN {X 0,Y 333.783,Z 321.382,A -85,B 0,C 180,E1 -14395.168,E2 -14395.168} C_VEL
LIN {X 0,Y 334.069,Z 321.363,A -85,B 0,C 180,E1 -14397.588,E2 -14397.588} C_VEL
LIN {X 0,Y 334.079,Z 321.361,A -85,B 0,C 180,E1 -14401.205,E2 -14401.205} C_VEL
LIN {X 0,Y 333.804,Z 321.38,A -85,B 0,C 180,E1 -14403.621,E2 -14403.621} C_VEL
LIN {X 0,Y 334.003,Z 321.356,A -85,B 0,C 180,E1 -14406.039,E2 -14406.039} C_VEL
LIN {X 0,Y 333.822,Z 321.402,A -85,B 0,C 180,E1 -14409.696,E2 -14409.696} C_VEL
LIN {X 0,Y 333.788,Z 321.392,A -85,B 0,C 180,E1 -14413.391,E2 -14413.391} C_VEL
LIN {X 0,Y 333.685,Z 321.407,A -85,B 0,C 180,E1 -14417.149,E2 -14417.149} C_VEL
LIN {X 0,Y 333.653,Z 321.423,A -85,B 0,C 180,E1 -14419.695,E2 -14419.695} C_VEL
LIN {X 0,Y 333.654,Z 321.404,A -85,B 0,C 180,E1 -14423.591,E2 -14423.591} C_VEL
LIN {X 0,Y 333.651,Z 321.417,A -85,B 0,C 180,E1 -14426.253,E2 -14426.253} C_VEL
LIN {X 0,Y 333.657,Z 321.414,A -85,B 0,C 180,E1 -14430.366,E2 -14430.366} C_VEL
LIN {X 0,Y 333.637,Z 321.422,A -85,B 0,C 180,E1 -14433.208,E2 -14433.208} C_VEL
LIN {X 0,Y 333.674,Z 321.413,A -85,B 0,C 180,E1 -14436.139,E2 -14436.139} C_VEL
LIN {X 0,Y 333.6,Z 321.426,A -85,B 0,C 180,E1 -14439.198,E2 -14439.198} C_VEL
LIN {X 0,Y 333.625,Z 321.419,A -85,B 0,C 180,E1 -14442.498,E2 -14442.498} C_VEL
LIN {X 0,Y 333.591,Z 321.429,A -85,B 0,C 180,E1 -14445.954,E2 -14445.954} C_VEL
LIN {X 0,Y 333.6,Z 321.427,A -85,B 0,C 180,E1 -14449.324,E2 -14449.324} C_VEL
LIN {X 0,Y 333.66,Z 321.424,A -85,B 0,C 180,E1 -14453.168,E2 -14453.168} C_VEL
LIN {X 0,Y 333.671,Z 321.418,A -85,B 0,C 180,E1 -14455.341,E2 -14455.341} C_VEL
LIN {X 0,Y 333.627,Z 321.428,A -85,B 0,C 180,E1 -14458.221,E2 -14458.221} C_VEL
LIN {X 0,Y 333.71,Z 321.612,A -85,B 0,C 180,E1 -14459.838,E2 -14459.838} C_VEL
LIN {X 0,Y 336.353,Z 334.27,A -85,B 0,C 180,E1 -14463.64,E2 -14463.64} C_VEL
LIN {X 0,Y 337.487,Z 341.424,A -85,B 0,C 180,E1 -14465.682,E2 -14465.682} C_VEL
LIN {X 0,Y 337.238,Z 344.527,A -85,B 0,C 180,E1 -14466.43,E2 -14466.43} C_VEL
LIN {X 0,Y 341.556,Z 369.535,A -85,B 0,C 180,E1 -14467.326,E2 -14467.326} C_VEL
LIN {X 0,Y 343.023,Z 379.669,A -85,B 0,C 180,E1 -14467.649,E2 -14467.649} C_VEL
LIN {X 0,Y 341.509,Z 451.18,A -85,B 0,C 180,E1 -14469.207,E2 -14469.207} C_VEL
LIN {X 0,Y 341.163,Z 460.752,A -85,B 0,C 180,E1 -14469.54,E2 -14469.54} C_VEL
LIN {X 0,Y 340.455,Z 470.588,A -85,B 0,C 180,E1 -14470.007,E2 -14470.007} C_VEL
LIN {X 0,Y 339.728,Z 480.871,A -85,B 0,C 180,E1 -14470.671,E2 -14470.671} C_VEL
LIN {X 0,Y 338.65,Z 491.51,A -85,B 0,C 180,E1 -14471.549,E2 -14471.549} C_VEL
LIN {X 0,Y 337.622,Z 501.485,A -85,B 0,C 180,E1 -14472.588,E2 -14472.588} C_VEL
LIN {X 0,Y 336.691,Z 509.803,A -85,B 0,C 180,E1 -14473.633,E2 -14473.633} C_VEL
LIN {X 0,Y 335.755,Z 517.803,A -85,B 0,C 180,E1 -14474.832,E2 -14474.832} C_VEL
LIN {X 0,Y 334.754,Z 526.085,A -85,B 0,C 180,E1 -14476.338,E2 -14476.338} C_VEL
LIN {X 0,Y 333.804,Z 532.974,A -85,B 0,C 180,E1 -14477.846,E2 -14477.846} C_VEL
LIN {X 0,Y 333.185,Z 538.736,A -85,B 0,C 180,E1 -14479.364,E2 -14479.364} C_VEL
LIN {X 0,Y 332.697,Z 543.521,A -85,B 0,C 180,E1 -14480.884,E2 -14480.884} C_VEL
LIN {X 0,Y 332.277,Z 548.094,A -85,B 0,C 180,E1 -14482.709,E2 -14482.709} C_VEL
LIN {X 0,Y 332.062,Z 550.795,A -85,B 0,C 180,E1 -14484.116,E2 -14484.116} C_VEL
LIN {X 0,Y 331.952,Z 554.02,A -85,B 0,C 180,E1 -14486.358,E2 -14486.358} C_VEL
LIN {X 0,Y 331.86,Z 555.775,A -85,B 0,C 180,E1 -14488.786,E2 -14488.786} C_VEL
LIN {X 0,Y 331.881,Z 556.092,A -85,B 0,C 180,E1 -14490,E2 -14490} C_VEL
LIN {X 0,Y 331.88,Z 555.516,A -85,B 0,C 180,E1 -14492.427,E2 -14492.427} C_VEL
LIN {X 0,Y 332.017,Z 553.214,A -85,B 0,C 180,E1 -14494.857,E2 -14494.857} C_VEL
LIN {X 0,Y 332.177,Z 550.442,A -85,B 0,C 180,E1 -14496.682,E2 -14496.682} C_VEL
LIN {X 0,Y 332.568,Z 546.641,A -85,B 0,C 180,E1 -14498.507,E2 -14498.507} C_VEL
LIN {X 0,Y 333.141,Z 541.709,A -85,B 0,C 180,E1 -14500.33,E2 -14500.33} C_VEL
LIN {X 0,Y 333.807,Z 536.669,A -85,B 0,C 180,E1 -14501.846,E2 -14501.846} C_VEL
LIN {X 0,Y 334.741,Z 530.603,A -85,B 0,C 180,E1 -14503.353,E2 -14503.353} C_VEL
LIN {X 0,Y 335.817,Z 523.295,A -85,B 0,C 180,E1 -14504.855,E2 -14504.855} C_VEL
LIN {X 0,Y 336.889,Z 514.556,A -85,B 0,C 180,E1 -14506.338,E2 -14506.338} C_VEL
LIN {X 0,Y 338.069,Z 505.928,A -85,B 0,C 180,E1 -14507.544,E2 -14507.544} C_VEL
LIN {X 0,Y 339.212,Z 497.04,A -85,B 0,C 180,E1 -14508.575,E2 -14508.575} C_VEL
LIN {X 0,Y 340.523,Z 486.008,A -85,B 0,C 180,E1 -14509.596,E2 -14509.596} C_VEL
LIN {X 0,Y 341.423,Z 476.163,A -85,B 0,C 180,E1 -14510.326,E2 -14510.326} C_VEL
LIN {X 0,Y 342.396,Z 464.429,A -85,B 0,C 180,E1 -14510.972,E2 -14510.972} C_VEL
LIN {X 0,Y 343.035,Z 454.564,A -85,B 0,C 180,E1 -14511.364,E2 -14511.364} C_VEL
LIN {X 0,Y 343.553,Z 435.85,A -85,B 0,C 180,E1 -14511.827,E2 -14511.827} C_VEL
LIN {X 0,Y 344.726,Z 379.499,A -85,B 0,C 180,E1 -14513.047,E2 -14513.047} C_VEL
LIN {X 0,Y 341.139,Z 358.381,A -85,B 0,C 180,E1 -14513.826,E2 -14513.826} C_VEL
LIN {X 0,Y 338.175,Z 344.261,A -85,B 0,C 180,E1 -14514.439,E2 -14514.439} C_VEL
LIN {X 0,Y 338.14,Z 343.367,A -85,B 0,C 180,E1 -14514.562,E2 -14514.562} C_VEL
LIN {X 0,Y 336.822,Z 335.705,A -85,B 0,C 180,E1 -14516.716,E2 -14516.716} C_VEL
LIN {X 0,Y 334.223,Z 323.709,A -85,B 0,C 180,E1 -14520.309,E2 -14520.309} C_VEL
LIN {X 0,Y 333.677,Z 321.454,A -85,B 0,C 180,E1 -14521.109,E2 -14521.109} C_VEL
LIN {X 0,Y 333.683,Z 321.418,A -85,B 0,C 180,E1 -14524.774,E2 -14524.774} C_VEL
LIN {X 0,Y 333.65,Z 321.421,A -85,B 0,C 180,E1 -14527.651,E2 -14527.651} C_VEL
LIN {X 0,Y 333.643,Z 321.414,A -85,B 0,C 180,E1 -14530.768,E2 -14530.768} C_VEL
LIN {X 0,Y 333.591,Z 321.43,A -85,B 0,C 180,E1 -14534.251,E2 -14534.251} C_VEL
LIN {X 0,Y 333.64,Z 321.424,A -85,B 0,C 180,E1 -14537.619,E2 -14537.619} C_VEL
LIN {X 0,Y 333.651,Z 321.421,A -85,B 0,C 180,E1 -14541.202,E2 -14541.202} C_VEL
LIN {X 0,Y 333.675,Z 321.42,A -85,B 0,C 180,E1 -14543.861,E2 -14543.861} C_VEL
LIN {X 0,Y 333.645,Z 321.423,A -85,B 0,C 180,E1 -14547.413,E2 -14547.413} C_VEL
LIN {X 0,Y 333.689,Z 321.417,A -85,B 0,C 180,E1 -14551.026,E2 -14551.026} C_VEL
LIN {X 0,Y 333.735,Z 321.409,A -85,B 0,C 180,E1 -14553.754,E2 -14553.754} C_VEL
LIN {X 0,Y 333.719,Z 321.41,A -85,B 0,C 180,E1 -14557.914,E2 -14557.914} C_VEL
LIN {X 0,Y 333.795,Z 321.397,A -85,B 0,C 180,E1 -14561.59,E2 -14561.59} C_VEL
LIN {X 0,Y 333.809,Z 321.396,A -85,B 0,C 180,E1 -14565.577,E2 -14565.577} C_VEL
LIN {X 0,Y 333.835,Z 321.399,A -85,B 0,C 180,E1 -14569.078,E2 -14569.078} C_VEL
LIN {X 0,Y 334.028,Z 321.375,A -85,B 0,C 180,E1 -14572.748,E2 -14572.748} C_VEL
LIN {X 0,Y 333.812,Z 321.396,A -85,B 0,C 180,E1 -14575.169,E2 -14575.169} C_VEL
LIN {X 0,Y 334.108,Z 321.363,A -85,B 0,C 180,E1 -14577.589,E2 -14577.589} C_VEL
LIN {X 0,Y 334.249,Z 321.343,A -85,B 0,C 180,E1 -14580,E2 -14580} C_VEL
LIN {X 0,Y 334.108,Z 321.366,A -85,B 0,C 180,E1 -14582.411,E2 -14582.411} C_VEL
LIN {X 0,Y 334.027,Z 321.377,A -85,B 0,C 180,E1 -14587.253,E2 -14587.253} C_VEL
LIN {X 0,Y 333.835,Z 321.401,A -85,B 0,C 180,E1 -14590.922,E2 -14590.922} C_VEL
LIN {X 0,Y 333.809,Z 321.403,A -85,B 0,C 180,E1 -14594.634,E2 -14594.634} C_VEL
LIN {X 0,Y 333.797,Z 321.401,A -85,B 0,C 180,E1 -14598.655,E2 -14598.655} C_VEL
LIN {X 0,Y 333.657,Z 321.422,A -85,B 0,C 180,E1 -14602.281,E2 -14602.281} C_VEL
LIN {X 0,Y 333.709,Z 321.417,A -85,B 0,C 180,E1 -14605.097,E2 -14605.097} C_VEL
LIN {X 0,Y 333.686,Z 321.417,A -85,B 0,C 180,E1 -14608.975,E2 -14608.975} C_VEL
LIN {X 0,Y 333.644,Z 321.426,A -85,B 0,C 180,E1 -14612.587,E2 -14612.587} C_VEL
LIN {X 0,Y 333.678,Z 321.417,A -85,B 0,C 180,E1 -14616.139,E2 -14616.139} C_VEL
LIN {X 0,Y 333.72,Z 321.608,A -85,B 0,C 180,E1 -14617.389,E2 -14617.389} C_VEL
LIN {X 0,Y 336.019,Z 331.632,A -85,B 0,C 180,E1 -14620.42,E2 -14620.42} C_VEL
LIN {X 0,Y 336.863,Z 335.636,A -85,B 0,C 180,E1 -14621.484,E2 -14621.484} C_VEL
LIN {X 0,Y 340.947,Z 346.222,A -85,B 0,C 180,E1 -14622.111,E2 -14622.111} C_VEL
LIN {X 0,Y 344.99,Z 366.642,A -85,B 0,C 180,E1 -14622.918,E2 -14622.918} C_VEL
LIN {X 0,Y 343.231,Z 440.817,A -85,B 0,C 180,E1 -14624.535,E2 -14624.535} C_VEL
LIN {X 0,Y 342.748,Z 451.07,A -85,B 0,C 180,E1 -14624.871,E2 -14624.871} C_VEL
LIN {X 0,Y 342.14,Z 461.758,A -85,B 0,C 180,E1 -14625.392,E2 -14625.392} C_VEL
LIN {X 0,Y 341.263,Z 471.986,A -85,B 0,C 180,E1 -14626.05,E2 -14626.05} C_VEL
LIN {X 0,Y 340.314,Z 481.946,A -85,B 0,C 180,E1 -14626.873,E2 -14626.873} C_VEL
LIN {X 0,Y 339.172,Z 491.661,A -85,B 0,C 180,E1 -14627.869,E2 -14627.869} C_VEL
LIN {X 0,Y 337.936,Z 501.191,A -85,B 0,C 180,E1 -14629.073,E2 -14629.073} C_VEL
LIN {X 0,Y 336.826,Z 508.879,A -85,B 0,C 180,E1 -14630.231,E2 -14630.231} C_VEL
LIN {X 0,Y 335.579,Z 517.589,A -85,B 0,C 180,E1 -14631.843,E2 -14631.843} C_VEL
LIN {X 0,Y 334.594,Z 524.526,A -85,B 0,C 180,E1 -14633.406,E2 -14633.406} C_VEL
LIN {X 0,Y 333.913,Z 529.211,A -85,B 0,C 180,E1 -14634.634,E2 -14634.634} C_VEL
LIN {X 0,Y 333.042,Z 535.486,A -85,B 0,C 180,E1 -14636.725,E2 -14636.725} C_VEL
LIN {X 0,Y 332.633,Z 538.903,A -85,B 0,C 180,E1 -14638.116,E2 -14638.116} C_VEL
LIN {X 0,Y 332.231,Z 542.633,A -85,B 0,C 180,E1 -14640.148,E2 -14640.148} C_VEL
LIN {X 0,Y 331.814,Z 545.647,A -85,B 0,C 180,E1 -14642.821,E2 -14642.821} C_VEL
LIN {X 0,Y 331.695,Z 546.245,A -85,B 0,C 180,E1 -14643.58,E2 -14643.58} C_VEL
LIN {X 0,Y 331.595,Z 546.875,A -85,B 0,C 180,E1 -14645.695,E2 -14645.695} C_VEL
LIN {X 0,Y 331.63,Z 546.397,A -85,B 0,C 180,E1 -14647.576,E2 -14647.576} C_VEL
LIN {X 0,Y 331.75,Z 545.406,A -85,B 0,C 180,E1 -14648.891,E2 -14648.891} C_VEL
LIN {X 0,Y 331.864,Z 544.053,A -85,B 0,C 180,E1 -14650.194,E2 -14650.194} C_VEL
LIN {X 0,Y 332.09,Z 542.293,A -85,B 0,C 180,E1 -14651.492,E2 -14651.492} C_VEL
LIN {X 0,Y 332.452,Z 538.614,A -85,B 0,C 180,E1 -14653.418,E2 -14653.418} C_VEL
LIN {X 0,Y 333.094,Z 532.395,A -85,B 0,C 180,E1 -14655.75,E2 -14655.75} C_VEL
LIN {X 0,Y 333.659,Z 527.485,A -85,B 0,C 180,E1 -14657.223,E2 -14657.223} C_VEL
LIN {X 0,Y 334.44,Z 521.132,A -85,B 0,C 180,E1 -14658.792,E2 -14658.792} C_VEL
LIN {X 0,Y 335.435,Z 513.423,A -85,B 0,C 180,E1 -14660.351,E2 -14660.351} C_VEL
LIN {X 0,Y 336.456,Z 505.086,A -85,B 0,C 180,E1 -14661.743,E2 -14661.743} C_VEL
LIN {X 0,Y 337.513,Z 496.172,A -85,B 0,C 180,E1 -14662.973,E2 -14662.973} C_VEL
LIN {X 0,Y 338.499,Z 486.784,A -85,B 0,C 180,E1 -14664.041,E2 -14664.041} C_VEL
LIN {X 0,Y 339.449,Z 476.75,A -85,B 0,C 180,E1 -14664.967,E2 -14664.967} C_VEL
LIN {X 0,Y 340.343,Z 466.614,A -85,B 0,C 180,E1 -14665.707,E2 -14665.707} C_VEL
LIN {X 0,Y 340.966,Z 456,A -85,B 0,C 180,E1 -14666.307,E2 -14666.307} C_VEL
LIN {X 0,Y 341.522,Z 445.838,A -85,B 0,C 180,E1 -14666.719,E2 -14666.719} C_VEL
LIN {X 0,Y 341.996,Z 429.396,A -85,B 0,C 180,E1 -14667.129,E2 -14667.129} C_VEL
LIN {X 0,Y 343.179,Z 365.76,A -85,B 0,C 180,E1 -14668.494,E2 -14668.494} C_VEL
LIN {X 0,Y 338.356,Z 340.66,A -85,B 0,C 180,E1 -14669.379,E2 -14669.379} C_VEL
LIN {X 0,Y 336.809,Z 335.92,A -85,B 0,C 180,E1 -14669.629,E2 -14669.629} C_VEL
LIN {X 0,Y 335.47,Z 328.612,A -85,B 0,C 180,E1 -14671.801,E2 -14671.801} C_VEL
LIN {X 0,Y 333.825,Z 321.454,A -85,B 0,C 180,E1 -14674.15,E2 -14674.15} C_VEL
LIN {X 0,Y 334.01,Z 321.374,A -85,B 0,C 180,E1 -14676.039,E2 -14676.039} C_VEL
LIN {X 0,Y 333.823,Z 321.405,A -85,B 0,C 180,E1 -14679.696,E2 -14679.696} C_VEL
LIN {X 0,Y 333.799,Z 321.404,A -85,B 0,C 180,E1 -14683.391,E2 -14683.391} C_VEL
LIN {X 0,Y 333.748,Z 321.41,A -85,B 0,C 180,E1 -14687.146,E2 -14687.146} C_VEL
LIN {X 0,Y 333.735,Z 321.406,A -85,B 0,C 180,E1 -14689.691,E2 -14689.691} C_VEL
LIN {X 0,Y 333.67,Z 321.412,A -85,B 0,C 180,E1 -14693.799,E2 -14693.799} C_VEL
LIN {X 0,Y 333.003,Z 321.504,A -85,B 0,C 180,E1 -14694.807,E2 -14694.807} C_VEL
LIN {X 0,Y 330.143,Z 321.862,A -85,B 0,C 180,E1 -14696.446,E2 -14696.446} C_VEL
LIN {X 0,Y 327.727,Z 322.153,A -85,B 0,C 180,E1 -14697.774,E2 -14697.774} C_VEL
LIN {X 0,Y 326.703,Z 322.278,A -85,B 0,C 180,E1 -14698.802,E2 -14698.802} C_VEL
LIN {X 0,Y 326.627,Z 322.29,A -85,B 0,C 180,E1 -14699.151,E2 -14699.151} C_VEL
LIN {X 0,Y 326.619,Z 322.295,A -85,B 0,C 180,E1 -14702.946,E2 -14702.946} C_VEL
LIN {X 0,Y 326.614,Z 322.289,A -85,B 0,C 180,E1 -14705.52,E2 -14705.52} C_VEL
LIN {X 0,Y 326.613,Z 322.297,A -85,B 0,C 180,E1 -14709.227,E2 -14709.227} C_VEL
LIN {X 0,Y 326.584,Z 322.294,A -85,B 0,C 180,E1 -14712.973,E2 -14712.973} C_VEL
LIN {X 0,Y 326.582,Z 322.3,A -85,B 0,C 180,E1 -14717.027,E2 -14717.027} C_VEL
LIN {X 0,Y 326.6,Z 322.277,A -85,B 0,C 180,E1 -14720.776,E2 -14720.776} C_VEL
LIN {X 0,Y 326.614,Z 322.296,A -85,B 0,C 180,E1 -14724.48,E2 -14724.48} C_VEL
LIN {X 0,Y 326.61,Z 322.293,A -85,B 0,C 180,E1 -14727.455,E2 -14727.455} C_VEL
LIN {X 0,Y 326.619,Z 322.266,A -85,B 0,C 180,E1 -14730.337,E2 -14730.337} C_VEL
LIN {X 0,Y 326.652,Z 322.293,A -85,B 0,C 180,E1 -14734.641,E2 -14734.641} C_VEL
LIN {X 0,Y 326.622,Z 322.29,A -85,B 0,C 180,E1 -14738.543,E2 -14738.543} C_VEL
LIN {X 0,Y 326.709,Z 322.253,A -85,B 0,C 180,E1 -14741.175,E2 -14741.175} C_VEL
LIN {X 0,Y 326.765,Z 322.275,A -85,B 0,C 180,E1 -14745.433,E2 -14745.433} C_VEL
LIN {X 0,Y 326.76,Z 322.279,A -85,B 0,C 180,E1 -14748.838,E2 -14748.838} C_VEL
LIN {X 0,Y 326.915,Z 322.232,A -85,B 0,C 180,E1 -14752.589,E2 -14752.589} C_VEL
LIN {X 0,Y 326.752,Z 322.258,A -85,B 0,C 180,E1 -14755.064,E2 -14755.064} C_VEL
LIN {X 0,Y 327.012,Z 322.242,A -85,B 0,C 180,E1 -14757.536,E2 -14757.536} C_VEL
LIN {X 0,Y 327.047,Z 322.237,A -85,B 0,C 180,E1 -14761.231,E2 -14761.231} C_VEL
LIN {X 0,Y 326.753,Z 322.258,A -85,B 0,C 180,E1 -14763.699,E2 -14763.699} C_VEL
LIN {X 0,Y 326.959,Z 322.234,A -85,B 0,C 180,E1 -14766.169,E2 -14766.169} C_VEL
LIN {X 0,Y 326.784,Z 322.277,A -85,B 0,C 180,E1 -14769.907,E2 -14769.907} C_VEL
LIN {X 0,Y 326.744,Z 322.264,A -85,B 0,C 180,E1 -14773.686,E2 -14773.686} C_VEL
LIN {X 0,Y 326.632,Z 322.288,A -85,B 0,C 180,E1 -14777.531,E2 -14777.531} C_VEL
LIN {X 0,Y 326.608,Z 322.303,A -85,B 0,C 180,E1 -14780.138,E2 -14780.138} C_VEL
LIN {X 0,Y 326.629,Z 322.278,A -85,B 0,C 180,E1 -14784.13,E2 -14784.13} C_VEL
LIN {X 0,Y 326.599,Z 322.3,A -85,B 0,C 180,E1 -14788.082,E2 -14788.082} C_VEL
LIN {X 0,Y 326.572,Z 322.292,A -85,B 0,C 180,E1 -14791.097,E2 -14791.097} C_VEL
LIN {X 0,Y 326.607,Z 322.3,A -85,B 0,C 180,E1 -14794.019,E2 -14794.019} C_VEL
LIN {X 0,Y 326.622,Z 322.289,A -85,B 0,C 180,E1 -14797.237,E2 -14797.237} C_VEL
LIN {X 0,Y 326.542,Z 322.306,A -85,B 0,C 180,E1 -14801.124,E2 -14801.124} C_VEL
LIN {X 0,Y 326.557,Z 322.302,A -85,B 0,C 180,E1 -14803.526,E2 -14803.526} C_VEL
LIN {X 0,Y 326.57,Z 322.305,A -85,B 0,C 180,E1 -14807.029,E2 -14807.029} C_VEL
LIN {X 0,Y 326.58,Z 322.303,A -85,B 0,C 180,E1 -14811.385,E2 -14811.385} C_VEL
LIN {X 0,Y 326.616,Z 322.302,A -85,B 0,C 180,E1 -14814.851,E2 -14814.851} C_VEL
LIN {X 0,Y 326.606,Z 322.299,A -85,B 0,C 180,E1 -14817.455,E2 -14817.455} C_VEL
LIN {X 0,Y 326.602,Z 322.386,A -85,B 0,C 180,E1 -14819.399,E2 -14819.399} C_VEL
LIN {X 0,Y 328.806,Z 332.763,A -85,B 0,C 180,E1 -14822.642,E2 -14822.642} C_VEL
LIN {X 0,Y 330.532,Z 342.51,A -85,B 0,C 180,E1 -14825.505,E2 -14825.505} C_VEL
LIN {X 0,Y 330.445,Z 344.541,A -85,B 0,C 180,E1 -14825.965,E2 -14825.965} C_VEL
LIN {X 0,Y 335.833,Z 375.756,A -85,B 0,C 180,E1 -14827.097,E2 -14827.097} C_VEL
LIN {X 0,Y 336.399,Z 380.067,A -85,B 0,C 180,E1 -14827.234,E2 -14827.234} C_VEL
LIN {X 0,Y 334.826,Z 451.117,A -85,B 0,C 180,E1 -14828.812,E2 -14828.812} C_VEL
LIN {X 0,Y 334.422,Z 460.669,A -85,B 0,C 180,E1 -14829.148,E2 -14829.148} C_VEL
LIN {X 0,Y 333.672,Z 471.107,A -85,B 0,C 180,E1 -14829.663,E2 -14829.663} C_VEL
LIN {X 0,Y 333.007,Z 480.313,A -85,B 0,C 180,E1 -14830.265,E2 -14830.265} C_VEL
LIN {X 0,Y 331.921,Z 491.045,A -85,B 0,C 180,E1 -14831.162,E2 -14831.162} C_VEL
LIN {X 0,Y 330.827,Z 501.084,A -85,B 0,C 180,E1 -14832.219,E2 -14832.219} C_VEL
LIN {X 0,Y 329.799,Z 509.861,A -85,B 0,C 180,E1 -14833.344,E2 -14833.344} C_VEL
LIN {X 0,Y 328.89,Z 517.53,A -85,B 0,C 180,E1 -14834.514,E2 -14834.514} C_VEL
LIN {X 0,Y 327.84,Z 525.814,A -85,B 0,C 180,E1 -14836.044,E2 -14836.044} C_VEL
LIN {X 0,Y 326.838,Z 532.733,A -85,B 0,C 180,E1 -14837.583,E2 -14837.583} C_VEL
LIN {X 0,Y 326.055,Z 539.486,A -85,B 0,C 180,E1 -14839.443,E2 -14839.443} C_VEL
LIN {X 0,Y 325.651,Z 543.319,A -85,B 0,C 180,E1 -14840.685,E2 -14840.685} C_VEL
LIN {X 0,Y 325.207,Z 547.917,A -85,B 0,C 180,E1 -14842.55,E2 -14842.55} C_VEL
LIN {X 0,Y 324.975,Z 550.938,A -85,B 0,C 180,E1 -14844.154,E2 -14844.154} C_VEL
LIN {X 0,Y 324.86,Z 553.879,A -85,B 0,C 180,E1 -14846.279,E2 -14846.279} C_VEL
LIN {X 0,Y 324.772,Z 555.667,A -85,B 0,C 180,E1 -14848.76,E2 -14848.76} C_VEL
LIN {X 0,Y 324.789,Z 555.983,A -85,B 0,C 180,E1 -14850,E2 -14850} C_VEL
LIN {X 0,Y 324.802,Z 555.44,A -85,B 0,C 180,E1 -14852.48,E2 -14852.48} C_VEL
LIN {X 0,Y 324.927,Z 553.158,A -85,B 0,C 180,E1 -14854.963,E2 -14854.963} C_VEL
LIN {X 0,Y 325.116,Z 550.403,A -85,B 0,C 180,E1 -14856.828,E2 -14856.828} C_VEL
LIN {X 0,Y 325.521,Z 546.623,A -85,B 0,C 180,E1 -14858.692,E2 -14858.692} C_VEL
LIN {X 0,Y 326.155,Z 541.717,A -85,B 0,C 180,E1 -14860.554,E2 -14860.554} C_VEL
LIN {X 0,Y 326.839,Z 536.707,A -85,B 0,C 180,E1 -14862.102,E2 -14862.102} C_VEL
LIN {X 0,Y 327.84,Z 530.678,A -85,B 0,C 180,E1 -14863.639,E2 -14863.639} C_VEL
LIN {X 0,Y 328.956,Z 523.412,A -85,B 0,C 180,E1 -14865.172,E2 -14865.172} C_VEL
LIN {X 0,Y 330.133,Z 514.424,A -85,B 0,C 180,E1 -14866.727,E2 -14866.727} C_VEL
LIN {X 0,Y 331.311,Z 506.138,A -85,B 0,C 180,E1 -14867.914,E2 -14867.914} C_VEL
LIN {X 0,Y 332.668,Z 495.822,A -85,B 0,C 180,E1 -14869.114,E2 -14869.114} C_VEL
LIN {X 0,Y 333.863,Z 486.378,A -85,B 0,C 180,E1 -14870.003,E2 -14870.003} C_VEL
LIN {X 0,Y 334.928,Z 475.467,A -85,B 0,C 180,E1 -14870.818,E2 -14870.818} C_VEL
LIN {X 0,Y 335.804,Z 465.161,A -85,B 0,C 180,E1 -14871.404,E2 -14871.404} C_VEL
LIN {X 0,Y 336.516,Z 454.487,A -85,B 0,C 180,E1 -14871.839,E2 -14871.839} C_VEL
LIN {X 0,Y 337.052,Z 436.257,A -85,B 0,C 180,E1 -14872.3,E2 -14872.3} C_VEL
LIN {X 0,Y 338.305,Z 380.478,A -85,B 0,C 180,E1 -14873.528,E2 -14873.528} C_VEL
LIN {X 0,Y 334.719,Z 359.275,A -85,B 0,C 180,E1 -14874.341,E2 -14874.341} C_VEL
LIN {X 0,Y 331.618,Z 345.314,A -85,B 0,C 180,E1 -14874.958,E2 -14874.958} C_VEL
LIN {X 0,Y 331.14,Z 343.551,A -85,B 0,C 180,E1 -14875.117,E2 -14875.117} C_VEL
LIN {X 0,Y 329.187,Z 333.571,A -85,B 0,C 180,E1 -14878.014,E2 -14878.014} C_VEL
LIN {X 0,Y 326.961,Z 323.846,A -85,B 0,C 180,E1 -14881.056,E2 -14881.056} C_VEL
LIN {X 0,Y 326.603,Z 322.328,A -85,B 0,C 180,E1 -14881.658,E2 -14881.658} C_VEL
LIN {X 0,Y 326.611,Z 322.302,A -85,B 0,C 180,E1 -14885.52,E2 -14885.52} C_VEL
LIN {X 0,Y 326.609,Z 322.295,A -85,B 0,C 180,E1 -14889.227,E2 -14889.227} C_VEL
LIN {X 0,Y 326.573,Z 322.305,A -85,B 0,C 180,E1 -14892.972,E2 -14892.972} C_VEL
LIN {X 0,Y 326.574,Z 322.305,A -85,B 0,C 180,E1 -14897.028,E2 -14897.028} C_VEL
LIN {X 0,Y 326.61,Z 322.298,A -85,B 0,C 180,E1 -14900.773,E2 -14900.773} C_VEL
LIN {X 0,Y 326.611,Z 322.294,A -85,B 0,C 180,E1 -14904.481,E2 -14904.481} C_VEL
LIN {X 0,Y 326.609,Z 322.299,A -85,B 0,C 180,E1 -14907.456,E2 -14907.456} C_VEL
LIN {X 0,Y 326.647,Z 322.297,A -85,B 0,C 180,E1 -14910.34,E2 -14910.34} C_VEL
LIN {X 0,Y 326.69,Z 322.291,A -85,B 0,C 180,E1 -14914.517,E2 -14914.517} C_VEL
LIN {X 0,Y 326.647,Z 322.293,A -85,B 0,C 180,E1 -14918.546,E2 -14918.546} C_VEL
LIN {X 0,Y 326.744,Z 322.276,A -85,B 0,C 180,E1 -14921.178,E2 -14921.178} C_VEL
LIN {X 0,Y 326.763,Z 322.275,A -85,B 0,C 180,E1 -14925.433,E2 -14925.433} C_VEL
LIN {X 0,Y 326.771,Z 322.279,A -85,B 0,C 180,E1 -14928.839,E2 -14928.839} C_VEL
LIN {X 0,Y 326.979,Z 322.254,A -85,B 0,C 180,E1 -14932.591,E2 -14932.591} C_VEL
LIN {X 0,Y 326.779,Z 322.272,A -85,B 0,C 180,E1 -14935.065,E2 -14935.065} C_VEL
LIN {X 0,Y 327.049,Z 322.243,A -85,B 0,C 180,E1 -14937.537,E2 -14937.537} C_VEL
LIN {X 0,Y 327.2,Z 322.22,A -85,B 0,C 180,E1 -14940,E2 -14940} C_VEL
LIN {X 0,Y 327.049,Z 322.246,A -85,B 0,C 180,E1 -14942.464,E2 -14942.464} C_VEL
LIN {X 0,Y 326.974,Z 322.251,A -85,B 0,C 180,E1 -14946.638,E2 -14946.638} C_VEL
LIN {X 0,Y 326.815,Z 322.274,A -85,B 0,C 180,E1 -14949.906,E2 -14949.906} C_VEL
LIN {X 0,Y 326.76,Z 322.281,A -85,B 0,C 180,E1 -14953.686,E2 -14953.686} C_VEL
LIN {X 0,Y 326.701,Z 322.29,A -85,B 0,C 180,E1 -14957.528,E2 -14957.528} C_VEL
LIN {X 0,Y 326.659,Z 322.295,A -85,B 0,C 180,E1 -14960.135,E2 -14960.135} C_VEL
LIN {X 0,Y 326.645,Z 322.296,A -85,B 0,C 180,E1 -14964.13,E2 -14964.13} C_VEL
LIN {X 0,Y 326.643,Z 322.285,A -85,B 0,C 180,E1 -14968.252,E2 -14968.252} C_VEL
LIN {X 0,Y 326.59,Z 322.296,A -85,B 0,C 180,E1 -14971.096,E2 -14971.096} C_VEL
LIN {X 0,Y 326.608,Z 322.295,A -85,B 0,C 180,E1 -14974.02,E2 -14974.02} C_VEL
LIN {X 0,Y 326.657,Z 322.468,A -85,B 0,C 180,E1 -14976.851,E2 -14976.851} C_VEL
LIN {X 0,Y 329.195,Z 333.345,A -85,B 0,C 180,E1 -14980.227,E2 -14980.227} C_VEL
LIN {X 0,Y 329.698,Z 335.741,A -85,B 0,C 180,E1 -14980.855,E2 -14980.855} C_VEL
LIN {X 0,Y 334.833,Z 348.563,A -85,B 0,C 180,E1 -14981.651,E2 -14981.651} C_VEL
LIN {X 0,Y 338.571,Z 367.682,A -85,B 0,C 180,E1 -14982.433,E2 -14982.433} C_VEL
LIN {X 0,Y 336.666,Z 442.093,A -85,B 0,C 180,E1 -14984.091,E2 -14984.091} C_VEL
LIN {X 0,Y 336.162,Z 451.919,A -85,B 0,C 180,E1 -14984.431,E2 -14984.431} C_VEL
LIN {X 0,Y 335.525,Z 462.62,A -85,B 0,C 180,E1 -14984.976,E2 -14984.976} C_VEL
LIN {X 0,Y 334.588,Z 472.922,A -85,B 0,C 180,E1 -14985.665,E2 -14985.665} C_VEL
LIN {X 0,Y 333.74,Z 481.649,A -85,B 0,C 180,E1 -14986.397,E2 -14986.397} C_VEL
LIN {X 0,Y 332.524,Z 491.691,A -85,B 0,C 180,E1 -14987.442,E2 -14987.442} C_VEL
LIN {X 0,Y 331.214,Z 501.289,A -85,B 0,C 180,E1 -14988.677,E2 -14988.677} C_VEL
LIN {X 0,Y 330.029,Z 509.001,A -85,B 0,C 180,E1 -14989.86,E2 -14989.86} C_VEL
LIN {X 0,Y 328.889,Z 516.83,A -85,B 0,C 180,E1 -14991.315,E2 -14991.315} C_VEL
LIN {X 0,Y 327.677,Z 524.615,A -85,B 0,C 180,E1 -14993.091,E2 -14993.091} C_VEL
LIN {X 0,Y 326.878,Z 529.824,A -85,B 0,C 180,E1 -14994.514,E2 -14994.514} C_VEL
LIN {X 0,Y 326.29,Z 534.203,A -85,B 0,C 180,E1 -14995.943,E2 -14995.943} C_VEL
LIN {X 0,Y 325.556,Z 539.317,A -85,B 0,C 180,E1 -14998.069,E2 -14998.069} C_VEL
LIN {X 0,Y 325.12,Z 542.995,A -85,B 0,C 180,E1 -15000.186,E2 -15000.186} C_VEL
LIN {X 0,Y 324.847,Z 544.8,A -85,B 0,C 180,E1 -15001.578,E2 -15001.578} C_VEL
LIN {X 0,Y 324.687,Z 545.938,A -85,B 0,C 180,E1 -15002.964,E2 -15002.964} C_VEL
LIN {X 0,Y 324.492,Z 546.944,A -85,B 0,C 180,E1 -15005.458,E2 -15005.458} C_VEL
LIN {X 0,Y 324.498,Z 546.64,A -85,B 0,C 180,E1 -15007.055,E2 -15007.055} C_VEL
LIN {X 0,Y 324.732,Z 544.811,A -85,B 0,C 180,E1 -15009.74,E2 -15009.74} C_VEL
LIN {X 0,Y 325.1,Z 541.586,A -85,B 0,C 180,E1 -15012.025,E2 -15012.025} C_VEL
LIN {X 0,Y 325.404,Z 538.358,A -85,B 0,C 180,E1 -15013.694,E2 -15013.694} C_VEL
LIN {X 0,Y 325.929,Z 533.674,A -85,B 0,C 180,E1 -15015.543,E2 -15015.543} C_VEL
LIN {X 0,Y 326.594,Z 528.23,A -85,B 0,C 180,E1 -15017.258,E2 -15017.258} C_VEL
LIN {X 0,Y 327.371,Z 522.015,A -85,B 0,C 180,E1 -15018.86,E2 -15018.86} C_VEL
LIN {X 0,Y 328.389,Z 514.459,A -85,B 0,C 180,E1 -15020.453,E2 -15020.453} C_VEL
LIN {X 0,Y 329.557,Z 505.248,A -85,B 0,C 180,E1 -15022.032,E2 -15022.032} C_VEL
LIN {X 0,Y 330.653,Z 496.345,A -85,B 0,C 180,E1 -15023.287,E2 -15023.287} C_VEL
LIN {X 0,Y 331.65,Z 487.301,A -85,B 0,C 180,E1 -15024.343,E2 -15024.343} C_VEL
LIN {X 0,Y 332.656,Z 477.147,A -85,B 0,C 180,E1 -15025.304,E2 -15025.304} C_VEL
LIN {X 0,Y 333.587,Z 466.851,A -85,B 0,C 180,E1 -15026.074,E2 -15026.074} C_VEL
LIN {X 0,Y 334.256,Z 456.256,A -85,B 0,C 180,E1 -15026.685,E2 -15026.685} C_VEL
LIN {X 0,Y 334.879,Z 444.868,A -85,B 0,C 180,E1 -15027.143,E2 -15027.143} C_VEL
LIN {X 0,Y 335.333,Z 428.186,A -85,B 0,C 180,E1 -15027.56,E2 -15027.56} C_VEL
LIN {X 0,Y 336.511,Z 366.5,A -85,B 0,C 180,E1 -15028.906,E2 -15028.906} C_VEL
LIN {X 0,Y 331.924,Z 342.752,A -85,B 0,C 180,E1 -15029.769,E2 -15029.769} C_VEL
LIN {X 0,Y 329.713,Z 336.096,A -85,B 0,C 180,E1 -15030.115,E2 -15030.115} C_VEL
LIN {X 0,Y 328.6,Z 330.346,A -85,B 0,C 180,E1 -15031.839,E2 -15031.839} C_VEL
LIN {X 0,Y 326.785,Z 322.33,A -85,B 0,C 180,E1 -15034.51,E2 -15034.51} C_VEL
LIN {X 0,Y 326.984,Z 322.25,A -85,B 0,C 180,E1 -15036.169,E2 -15036.169} C_VEL
LIN {X 0,Y 326.785,Z 322.28,A -85,B 0,C 180,E1 -15039.907,E2 -15039.907} C_VEL
LIN {X 0,Y 326.761,Z 322.284,A -85,B 0,C 180,E1 -15043.685,E2 -15043.685} C_VEL
LIN {X 0,Y 326.701,Z 322.29,A -85,B 0,C 180,E1 -15047.528,E2 -15047.528} C_VEL
LIN {X 0,Y 326.661,Z 322.291,A -85,B 0,C 180,E1 -15050.135,E2 -15050.135} C_VEL
LIN {X 0,Y 326.652,Z 322.288,A -85,B 0,C 180,E1 -15054.129,E2 -15054.129} C_VEL
LIN {X 0,Y 326.685,Z 322.287,A -85,B 0,C 180,E1 -15056.858,E2 -15056.858} C_VEL
LIN {X 0,Y 326.627,Z 322.29,A -85,B 0,C 180,E1 -15059.151,E2 -15059.151} C_VEL
LIN {X 0,Y 325.968,Z 322.379,A -85,B 0,C 180,E1 -15060.179,E2 -15060.179} C_VEL
LIN {X 0,Y 323.083,Z 322.737,A -85,B 0,C 180,E1 -15061.851,E2 -15061.851} C_VEL
LIN {X 0,Y 320.643,Z 323.035,A -85,B 0,C 180,E1 -15063.206,E2 -15063.206} C_VEL
LIN {X 0,Y 319.619,Z 323.154,A -85,B 0,C 180,E1 -15064.256,E2 -15064.256} C_VEL
LIN {X 0,Y 319.548,Z 323.162,A -85,B 0,C 180,E1 -15064.612,E2 -15064.612} C_VEL
LIN {X 0,Y 319.575,Z 323.179,A -85,B 0,C 180,E1 -15068.008,E2 -15068.008} C_VEL
LIN {X 0,Y 319.528,Z 323.163,A -85,B 0,C 180,E1 -15071.597,E2 -15071.597} C_VEL
LIN {X 0,Y 319.517,Z 323.185,A -85,B 0,C 180,E1 -15074.738,E2 -15074.738} C_VEL
LIN {X 0,Y 319.561,Z 323.175,A -85,B 0,C 180,E1 -15077.017,E2 -15077.017} C_VEL
LIN {X 0,Y 319.546,Z 323.154,A -85,B 0,C 180,E1 -15080.371,E2 -15080.371} C_VEL
LIN {X 0,Y 319.581,Z 323.172,A -85,B 0,C 180,E1 -15084.457,E2 -15084.457} C_VEL
LIN {X 0,Y 319.526,Z 323.168,A -85,B 0,C 180,E1 -15088.137,E2 -15088.137} C_VEL
LIN {X 0,Y 319.574,Z 323.147,A -85,B 0,C 180,E1 -15091.603,E2 -15091.603} C_VEL
LIN {X 0,Y 319.586,Z 323.171,A -85,B 0,C 180,E1 -15095.302,E2 -15095.302} C_VEL
LIN {X 0,Y 319.571,Z 323.175,A -85,B 0,C 180,E1 -15098.046,E2 -15098.046} C_VEL
